LIN {X 0,Y 573.181,Z 132.082,A -85,B 0,C 180,E1 -2286.055,E2 -2286.055} C_VEL
LIN {X 0,Y 573.23,Z 132.081,A -85,B 0,C 180,E1 -2288.703,E2 -2288.703} C_VEL
LIN {X 0,Y 573.201,Z 132.082,A -85,B 0,C 180,E1 -2291.46,E2 -2291.46} C_VEL
LIN {X 0,Y 573.219,Z 132.079,A -85,B 0,C 180,E1 -2294.336,E2 -2294.336} C_VEL
LIN {X 0,Y 573.214,Z 132.079,A -85,B 0,C 180,E1 -2297.362,E2 -2297.362} C_VEL
LIN {X 0,Y 573.229,Z 132.08,A -85,B 0,C 180,E1 -2300.391,E2 -2300.391} C_VEL
LIN {X 0,Y 573.231,Z 132.078,A -85,B 0,C 180,E1 -2303.076,E2 -2303.076} C_VEL
LIN {X 0,Y 573.248,Z 132.074,A -85,B 0,C 180,E1 -2305.67,E2 -2305.67} C_VEL
LIN {X 0,Y 573.227,Z 132.081,A -85,B 0,C 180,E1 -2308.184,E2 -2308.184} C_VEL
LIN {X 0,Y 573.219,Z 132.083,A -85,B 0,C 180,E1 -2310.632,E2 -2310.632} C_VEL
LIN {X 0,Y 573.207,Z 132.079,A -85,B 0,C 180,E1 -2313.515,E2 -2313.515} C_VEL
LIN {X 0,Y 573.201,Z 132.087,A -85,B 0,C 180,E1 -2316.133,E2 -2316.133} C_VEL
LIN {X 0,Y 573.238,Z 132.076,A -85,B 0,C 180,E1 -2318.714,E2 -2318.714} C_VEL
LIN {X 0,Y 573.199,Z 132.08,A -85,B 0,C 180,E1 -2321.411,E2 -2321.411} C_VEL
LIN {X 0,Y 573.21,Z 132.084,A -85,B 0,C 180,E1 -2324.351,E2 -2324.351} C_VEL
LIN {X 0,Y 573.206,Z 132.081,A -85,B 0,C 180,E1 -2326.529,E2 -2326.529} C_VEL
LIN {X 0,Y 573.261,Z 132.075,A -85,B 0,C 180,E1 -2329.403,E2 -2329.403} C_VEL
LIN {X 0,Y 573.225,Z 132.081,A -85,B 0,C 180,E1 -2332.249,E2 -2332.249} C_VEL
LIN {X 0,Y 573.288,Z 132.07,A -85,B 0,C 180,E1 -2335.077,E2 -2335.077} C_VEL
LIN {X 0,Y 573.313,Z 132.072,A -85,B 0,C 180,E1 -2337.893,E2 -2337.893} C_VEL
LIN {X 0,Y 573.322,Z 132.07,A -85,B 0,C 180,E1 -2340,E2 -2340} C_VEL
LIN {X 0,Y 573.287,Z 132.071,A -85,B 0,C 180,E1 -2342.811,E2 -2342.811} C_VEL
LIN {X 0,Y 573.284,Z 132.078,A -85,B 0,C 180,E1 -2345.628,E2 -2345.628} C_VEL
LIN {X 0,Y 573.285,Z 132.18,A -85,B 0,C 180,E1 -2348.371,E2 -2348.371} C_VEL
LIN {X 0,Y 573.5,Z 140.017,A -85,B 0,C 180,E1 -2349.701,E2 -2349.701} C_VEL
LIN {X 0,Y 573.378,Z 155.55,A -85,B 0,C 180,E1 -2352.386,E2 -2352.386} C_VEL
LIN {X 0,Y 573.294,Z 166.446,A -85,B 0,C 180,E1 -2354.231,E2 -2354.231} C_VEL
LIN {X 0,Y 574.098,Z 171.713,A -85,B 0,C 180,E1 -2354.317,E2 -2354.317} C_VEL
LIN {X 0,Y 573.971,Z 236.172,A -85,B 0,C 180,E1 -2355.126,E2 -2355.126} C_VEL
LIN {X 0,Y 573.349,Z 242.014,A -85,B 0,C 180,E1 -2355.185,E2 -2355.185} C_VEL
LIN {X 0,Y 567.678,Z 260.997,A -85,B 0,C 180,E1 -2355.294,E2 -2355.294} C_VEL
LIN {X 0,Y 566.978,Z 266.837,A -85,B 0,C 180,E1 -2355.355,E2 -2355.355} C_VEL
LIN {X 0,Y 566.881,Z 279.861,A -85,B 0,C 180,E1 -2355.598,E2 -2355.598} C_VEL
LIN {X 0,Y 566.804,Z 291.142,A -85,B 0,C 180,E1 -2355.923,E2 -2355.923} C_VEL
LIN {X 0,Y 566.703,Z 302.843,A -85,B 0,C 180,E1 -2356.388,E2 -2356.388} C_VEL
LIN {X 0,Y 566.554,Z 313.939,A -85,B 0,C 180,E1 -2356.973,E2 -2356.973} C_VEL
LIN {X 0,Y 566.407,Z 324.984,A -85,B 0,C 180,E1 -2357.698,E2 -2357.698} C_VEL
LIN {X 0,Y 566.246,Z 335.181,A -85,B 0,C 180,E1 -2358.545,E2 -2358.545} C_VEL
LIN {X 0,Y 566.193,Z 343.437,A -85,B 0,C 180,E1 -2359.374,E2 -2359.374} C_VEL
LIN {X 0,Y 566.095,Z 351.459,A -85,B 0,C 180,E1 -2360.342,E2 -2360.342} C_VEL
LIN {X 0,Y 565.998,Z 358.286,A -85,B 0,C 180,E1 -2361.364,E2 -2361.364} C_VEL
LIN {X 0,Y 565.939,Z 363.21,A -85,B 0,C 180,E1 -2362.257,E2 -2362.257} C_VEL
LIN {X 0,Y 565.912,Z 368.377,A -85,B 0,C 180,E1 -2363.416,E2 -2363.416} C_VEL
LIN {X 0,Y 565.916,Z 372.21,A -85,B 0,C 180,E1 -2364.572,E2 -2364.572} C_VEL
LIN {X 0,Y 565.839,Z 374.92,A -85,B 0,C 180,E1 -2365.768,E2 -2365.768} C_VEL
LIN {X 0,Y 565.863,Z 376.12,A -85,B 0,C 180,E1 -2366.588,E2 -2366.588} C_VEL
LIN {X 0,Y 565.834,Z 376.788,A -85,B 0,C 180,E1 -2367.359,E2 -2367.359} C_VEL
LIN {X 0,Y 565.835,Z 376.98,A -85,B 0,C 180,E1 -2368.163,E2 -2368.163} C_VEL
LIN {X 0,Y 565.849,Z 376.658,A -85,B 0,C 180,E1 -2368.973,E2 -2368.973} C_VEL
LIN {X 0,Y 565.874,Z 375.805,A -85,B 0,C 180,E1 -2369.788,E2 -2369.788} C_VEL
LIN {X 0,Y 565.882,Z 373.468,A -85,B 0,C 180,E1 -2371.024,E2 -2371.024} C_VEL
LIN {X 0,Y 565.886,Z 369.468,A -85,B 0,C 180,E1 -2372.378,E2 -2372.378} C_VEL
LIN {X 0,Y 565.954,Z 363.904,A -85,B 0,C 180,E1 -2373.694,E2 -2373.694} C_VEL
LIN {X 0,Y 565.987,Z 357.645,A -85,B 0,C 180,E1 -2374.834,E2 -2374.834} C_VEL
LIN {X 0,Y 566.077,Z 349.885,A -85,B 0,C 180,E1 -2375.951,E2 -2375.951} C_VEL
LIN {X 0,Y 566.18,Z 341.688,A -85,B 0,C 180,E1 -2376.905,E2 -2376.905} C_VEL
LIN {X 0,Y 566.332,Z 332.526,A -85,B 0,C 180,E1 -2377.788,E2 -2377.788} C_VEL
LIN {X 0,Y 566.413,Z 322.247,A -85,B 0,C 180,E1 -2378.583,E2 -2378.583} C_VEL
LIN {X 0,Y 566.564,Z 311.758,A -85,B 0,C 180,E1 -2379.245,E2 -2379.245} C_VEL
LIN {X 0,Y 566.74,Z 300.242,A -85,B 0,C 180,E1 -2379.816,E2 -2379.816} C_VEL
LIN {X 0,Y 566.816,Z 288.611,A -85,B 0,C 180,E1 -2380.249,E2 -2380.249} C_VEL
LIN {X 0,Y 566.93,Z 275.731,A -85,B 0,C 180,E1 -2380.589,E2 -2380.589} C_VEL
LIN {X 0,Y 567.007,Z 254.604,A -85,B 0,C 180,E1 -2380.891,E2 -2380.891} C_VEL
LIN {X 0,Y 567.047,Z 170.943,A -85,B 0,C 180,E1 -2381.957,E2 -2381.957} C_VEL
LIN {X 0,Y 566.278,Z 166.148,A -85,B 0,C 180,E1 -2382.045,E2 -2382.045} C_VEL
LIN {X 0,Y 566.471,Z 147.947,A -85,B 0,C 180,E1 -2385.255,E2 -2385.255} C_VEL
LIN {X 0,Y 566.53,Z 135.587,A -85,B 0,C 180,E1 -2387.46,E2 -2387.46} C_VEL
LIN {X 0,Y 566.211,Z 132.957,A -85,B 0,C 180,E1 -2387.984,E2 -2387.984} C_VEL
LIN {X 0,Y 566.208,Z 132.959,A -85,B 0,C 180,E1 -2390.725,E2 -2390.725} C_VEL
LIN {X 0,Y 566.183,Z 132.954,A -85,B 0,C 180,E1 -2393.428,E2 -2393.428} C_VEL
LIN {X 0,Y 566.201,Z 132.957,A -85,B 0,C 180,E1 -2396.268,E2 -2396.268} C_VEL
LIN {X 0,Y 566.181,Z 132.956,A -85,B 0,C 180,E1 -2398.926,E2 -2398.926} C_VEL
LIN {X 0,Y 566.147,Z 132.96,A -85,B 0,C 180,E1 -2401.853,E2 -2401.853} C_VEL
LIN {X 0,Y 566.184,Z 132.961,A -85,B 0,C 180,E1 -2404.249,E2 -2404.249} C_VEL
LIN {X 0,Y 566.162,Z 132.959,A -85,B 0,C 180,E1 -2406.722,E2 -2406.722} C_VEL
LIN {X 0,Y 566.189,Z 132.954,A -85,B 0,C 180,E1 -2408.901,E2 -2408.901} C_VEL
LIN {X 0,Y 566.167,Z 132.955,A -85,B 0,C 180,E1 -2411.17,E2 -2411.17} C_VEL
LIN {X 0,Y 566.172,Z 132.965,A -85,B 0,C 180,E1 -2414.151,E2 -2414.151} C_VEL
LIN {X 0,Y 566.171,Z 132.96,A -85,B 0,C 180,E1 -2416.358,E2 -2416.358} C_VEL
LIN {X 0,Y 566.216,Z 132.95,A -85,B 0,C 180,E1 -2419.269,E2 -2419.269} C_VEL
LIN {X 0,Y 566.192,Z 132.959,A -85,B 0,C 180,E1 -2422.152,E2 -2422.152} C_VEL
LIN {X 0,Y 566.253,Z 132.944,A -85,B 0,C 180,E1 -2425.015,E2 -2425.015} C_VEL
LIN {X 0,Y 566.281,Z 132.951,A -85,B 0,C 180,E1 -2427.866,E2 -2427.866} C_VEL
LIN {X 0,Y 566.289,Z 132.947,A -85,B 0,C 180,E1 -2429.999,E2 -2429.999} C_VEL
LIN {X 0,Y 566.241,Z 132.946,A -85,B 0,C 180,E1 -2432.845,E2 -2432.845} C_VEL
LIN {X 0,Y 566.24,Z 132.956,A -85,B 0,C 180,E1 -2435.698,E2 -2435.698} C_VEL
LIN {X 0,Y 566.188,Z 132.953,A -85,B 0,C 180,E1 -2438.566,E2 -2438.566} C_VEL
LIN {X 0,Y 566.196,Z 132.96,A -85,B 0,C 180,E1 -2441.455,E2 -2441.455} C_VEL
LIN {X 0,Y 566.179,Z 132.954,A -85,B 0,C 180,E1 -2444.482,E2 -2444.482} C_VEL
LIN {X 0,Y 566.16,Z 132.964,A -85,B 0,C 180,E1 -2447.332,E2 -2447.332} C_VEL
LIN {X 0,Y 566.176,Z 132.961,A -85,B 0,C 180,E1 -2449.581,E2 -2449.581} C_VEL
LIN {X 0,Y 566.148,Z 132.96,A -85,B 0,C 180,E1 -2451.864,E2 -2451.864} C_VEL
LIN {X 0,Y 566.18,Z 132.959,A -85,B 0,C 180,E1 -2455.02,E2 -2455.02} C_VEL
LIN {X 0,Y 566.16,Z 132.964,A -85,B 0,C 180,E1 -2457.341,E2 -2457.341} C_VEL
LIN {X 0,Y 566.146,Z 132.96,A -85,B 0,C 180,E1 -2459.771,E2 -2459.771} C_VEL
LIN {X 0,Y 566.19,Z 132.953,A -85,B 0,C 180,E1 -2462.427,E2 -2462.427} C_VEL
LIN {X 0,Y 566.159,Z 132.965,A -85,B 0,C 180,E1 -2464.986,E2 -2464.986} C_VEL
LIN {X 0,Y 566.188,Z 132.956,A -85,B 0,C 180,E1 -2467.461,E2 -2467.461} C_VEL
LIN {X 0,Y 566.202,Z 132.951,A -85,B 0,C 180,E1 -2470.199,E2 -2470.199} C_VEL
LIN {X 0,Y 566.174,Z 132.962,A -85,B 0,C 180,E1 -2473.056,E2 -2473.056} C_VEL
LIN {X 0,Y 566.152,Z 132.957,A -85,B 0,C 180,E1 -2476.053,E2 -2476.053} C_VEL
LIN {X 0,Y 566.146,Z 132.967,A -85,B 0,C 180,E1 -2478.857,E2 -2478.857} C_VEL
LIN {X 0,Y 566.193,Z 132.953,A -85,B 0,C 180,E1 -2481.443,E2 -2481.443} C_VEL
LIN {X 0,Y 566.133,Z 132.963,A -85,B 0,C 180,E1 -2484.305,E2 -2484.305} C_VEL
LIN {X 0,Y 566.186,Z 132.958,A -85,B 0,C 180,E1 -2486.895,E2 -2486.895} C_VEL
LIN {X 0,Y 566.154,Z 132.957,A -85,B 0,C 180,E1 -2489.405,E2 -2489.405} C_VEL
LIN {X 0,Y 566.135,Z 132.96,A -85,B 0,C 180,E1 -2491.853,E2 -2491.853} C_VEL
LIN {X 0,Y 566.182,Z 132.959,A -85,B 0,C 180,E1 -2494.249,E2 -2494.249} C_VEL
LIN {X 0,Y 566.149,Z 132.962,A -85,B 0,C 180,E1 -2496.722,E2 -2496.722} C_VEL
LIN {X 0,Y 566.183,Z 132.956,A -85,B 0,C 180,E1 -2498.901,E2 -2498.901} C_VEL
LIN {X 0,Y 566.175,Z 132.954,A -85,B 0,C 180,E1 -2501.171,E2 -2501.171} C_VEL
LIN {X 0,Y 566.162,Z 132.964,A -85,B 0,C 180,E1 -2504.151,E2 -2504.151} C_VEL
LIN {X 0,Y 566.155,Z 132.964,A -85,B 0,C 180,E1 -2506.358,E2 -2506.358} C_VEL
LIN {X 0,Y 566.204,Z 132.951,A -85,B 0,C 180,E1 -2509.269,E2 -2509.269} C_VEL
LIN {X 0,Y 566.179,Z 132.963,A -85,B 0,C 180,E1 -2512.152,E2 -2512.152} C_VEL
LIN {X 0,Y 566.243,Z 132.946,A -85,B 0,C 180,E1 -2515.016,E2 -2515.016} C_VEL
LIN {X 0,Y 566.273,Z 132.95,A -85,B 0,C 180,E1 -2517.866,E2 -2517.866} C_VEL
LIN {X 0,Y 566.278,Z 132.95,A -85,B 0,C 180,E1 -2520,E2 -2520} C_VEL
LIN {X 0,Y 566.23,Z 132.947,A -85,B 0,C 180,E1 -2522.846,E2 -2522.846} C_VEL
LIN {X 0,Y 566.23,Z 132.955,A -85,B 0,C 180,E1 -2525.698,E2 -2525.698} C_VEL
LIN {X 0,Y 566.177,Z 132.954,A -85,B 0,C 180,E1 -2528.566,E2 -2528.566} C_VEL
LIN {X 0,Y 566.184,Z 132.959,A -85,B 0,C 180,E1 -2531.455,E2 -2531.455} C_VEL
LIN {X 0,Y 566.194,Z 132.952,A -85,B 0,C 180,E1 -2534.494,E2 -2534.494} C_VEL
LIN {X 0,Y 566.148,Z 132.963,A -85,B 0,C 180,E1 -2537.333,E2 -2537.333} C_VEL
LIN {X 0,Y 566.165,Z 132.965,A -85,B 0,C 180,E1 -2539.582,E2 -2539.582} C_VEL
LIN {X 0,Y 566.138,Z 132.963,A -85,B 0,C 180,E1 -2541.865,E2 -2541.865} C_VEL
LIN {X 0,Y 566.144,Z 132.959,A -85,B 0,C 180,E1 -2544.183,E2 -2544.183} C_VEL
LIN {X 0,Y 566.163,Z 132.956,A -85,B 0,C 180,E1 -2546.652,E2 -2546.652} C_VEL
LIN {X 0,Y 566.138,Z 132.962,A -85,B 0,C 180,E1 -2549.772,E2 -2549.772} C_VEL
LIN {X 0,Y 566.183,Z 132.953,A -85,B 0,C 180,E1 -2552.428,E2 -2552.428} C_VEL
LIN {X 0,Y 566.151,Z 132.963,A -85,B 0,C 180,E1 -2554.987,E2 -2554.987} C_VEL
LIN {X 0,Y 566.181,Z 132.958,A -85,B 0,C 180,E1 -2557.462,E2 -2557.462} C_VEL
LIN {X 0,Y 566.159,Z 132.956,A -85,B 0,C 180,E1 -2560.203,E2 -2560.203} C_VEL
LIN {X 0,Y 566.141,Z 132.968,A -85,B 0,C 180,E1 -2563.06,E2 -2563.06} C_VEL
LIN {X 0,Y 566.148,Z 132.957,A -85,B 0,C 180,E1 -2566.054,E2 -2566.054} C_VEL
LIN {X 0,Y 566.136,Z 132.968,A -85,B 0,C 180,E1 -2568.858,E2 -2568.858} C_VEL
LIN {X 0,Y 566.165,Z 132.956,A -85,B 0,C 180,E1 -2571.636,E2 -2571.636} C_VEL
LIN {X 0,Y 566.126,Z 132.963,A -85,B 0,C 180,E1 -2574.306,E2 -2574.306} C_VEL
LIN {X 0,Y 566.158,Z 132.964,A -85,B 0,C 180,E1 -2576.895,E2 -2576.895} C_VEL
LIN {X 0,Y 566.145,Z 132.959,A -85,B 0,C 180,E1 -2579.406,E2 -2579.406} C_VEL
LIN {X 0,Y 566.137,Z 132.96,A -85,B 0,C 180,E1 -2581.854,E2 -2581.854} C_VEL
LIN {X 0,Y 566.172,Z 132.96,A -85,B 0,C 180,E1 -2584.25,E2 -2584.25} C_VEL
LIN {X 0,Y 566.157,Z 133.092,A -85,B 0,C 180,E1 -2586.833,E2 -2586.833} C_VEL
LIN {X 0,Y 566.94,Z 137.904,A -85,B 0,C 180,E1 -2587.593,E2 -2587.593} C_VEL
LIN {X 0,Y 566.776,Z 155.695,A -85,B 0,C 180,E1 -2590.252,E2 -2590.252} C_VEL
LIN {X 0,Y 566.546,Z 172.893,A -85,B 0,C 180,E1 -2592.782,E2 -2592.782} C_VEL
LIN {X 0,Y 566.404,Z 192.436,A -85,B 0,C 180,E1 -2595.632,E2 -2595.632} C_VEL
LIN {X 0,Y 566.421,Z 195.196,A -85,B 0,C 180,E1 -2595.999,E2 -2595.999} C_VEL
LIN {X 0,Y 567.174,Z 201.344,A -85,B 0,C 180,E1 -2596.097,E2 -2596.097} C_VEL
LIN {X 0,Y 566.965,Z 302.98,A -85,B 0,C 180,E1 -2597.404,E2 -2597.404} C_VEL
LIN {X 0,Y 566.839,Z 316.24,A -85,B 0,C 180,E1 -2597.719,E2 -2597.719} C_VEL
LIN {X 0,Y 566.741,Z 328.394,A -85,B 0,C 180,E1 -2598.149,E2 -2598.149} C_VEL
LIN {X 0,Y 566.602,Z 340.372,A -85,B 0,C 180,E1 -2598.72,E2 -2598.72} C_VEL
LIN {X 0,Y 566.439,Z 352.205,A -85,B 0,C 180,E1 -2599.456,E2 -2599.456} C_VEL
LIN {X 0,Y 566.325,Z 362.612,A -85,B 0,C 180,E1 -2600.266,E2 -2600.266} C_VEL
LIN {X 0,Y 566.207,Z 371.119,A -85,B 0,C 180,E1 -2601.075,E2 -2601.075} C_VEL
LIN {X 0,Y 566.112,Z 378.966,A -85,B 0,C 180,E1 -2601.972,E2 -2601.972} C_VEL
LIN {X 0,Y 566.003,Z 386.627,A -85,B 0,C 180,E1 -2603.047,E2 -2603.047} C_VEL
LIN {X 0,Y 566.004,Z 393.683,A -85,B 0,C 180,E1 -2604.3,E2 -2604.3} C_VEL
LIN {X 0,Y 565.933,Z 398.375,A -85,B 0,C 180,E1 -2605.371,E2 -2605.371} C_VEL
LIN {X 0,Y 565.927,Z 401.96,A -85,B 0,C 180,E1 -2606.441,E2 -2606.441} C_VEL
LIN {X 0,Y 565.877,Z 403.809,A -85,B 0,C 180,E1 -2607.153,E2 -2607.153} C_VEL
LIN {X 0,Y 565.846,Z 406.185,A -85,B 0,C 180,E1 -2608.577,E2 -2608.577} C_VEL
LIN {X 0,Y 565.839,Z 407,A -85,B 0,C 180,E1 -2610.001,E2 -2610.001} C_VEL
LIN {X 0,Y 565.846,Z 406.184,A -85,B 0,C 180,E1 -2611.424,E2 -2611.424} C_VEL
LIN {X 0,Y 565.878,Z 403.809,A -85,B 0,C 180,E1 -2612.848,E2 -2612.848} C_VEL
LIN {X 0,Y 565.926,Z 400.894,A -85,B 0,C 180,E1 -2613.917,E2 -2613.917} C_VEL
LIN {X 0,Y 565.878,Z 396.946,A -85,B 0,C 180,E1 -2614.988,E2 -2614.988} C_VEL
LIN {X 0,Y 566.002,Z 391.864,A -85,B 0,C 180,E1 -2616.059,E2 -2616.059} C_VEL
LIN {X 0,Y 566.041,Z 385.463,A -85,B 0,C 180,E1 -2617.133,E2 -2617.133} C_VEL
LIN {X 0,Y 566.134,Z 377.473,A -85,B 0,C 180,E1 -2618.208,E2 -2618.208} C_VEL
LIN {X 0,Y 566.229,Z 369.328,A -85,B 0,C 180,E1 -2619.106,E2 -2619.106} C_VEL
LIN {X 0,Y 566.348,Z 359.392,A -85,B 0,C 180,E1 -2620.005,E2 -2620.005} C_VEL
LIN {X 0,Y 566.536,Z 348.282,A -85,B 0,C 180,E1 -2620.808,E2 -2620.808} C_VEL
LIN {X 0,Y 566.614,Z 337.161,A -85,B 0,C 180,E1 -2621.447,E2 -2621.447} C_VEL
LIN {X 0,Y 566.746,Z 324.964,A -85,B 0,C 180,E1 -2621.989,E2 -2621.989} C_VEL
LIN {X 0,Y 566.918,Z 312.151,A -85,B 0,C 180,E1 -2622.394,E2 -2622.394} C_VEL
LIN {X 0,Y 566.994,Z 300.066,A -85,B 0,C 180,E1 -2622.642,E2 -2622.642} C_VEL
LIN {X 0,Y 567.043,Z 199.346,A -85,B 0,C 180,E1 -2623.932,E2 -2623.932} C_VEL
LIN {X 0,Y 566.385,Z 194.788,A -85,B 0,C 180,E1 -2624.026,E2 -2624.026} C_VEL
LIN {X 0,Y 566.532,Z 175.015,A -85,B 0,C 180,E1 -2626.896,E2 -2626.896} C_VEL
LIN {X 0,Y 566.723,Z 157.67,A -85,B 0,C 180,E1 -2629.424,E2 -2629.424} C_VEL
LIN {X 0,Y 566.911,Z 139.991,A -85,B 0,C 180,E1 -2632.025,E2 -2632.025} C_VEL
LIN {X 0,Y 566.504,Z 134.839,A -85,B 0,C 180,E1 -2632.799,E2 -2632.799} C_VEL
LIN {X 0,Y 566.155,Z 132.966,A -85,B 0,C 180,E1 -2633.093,E2 -2633.093} C_VEL
LIN {X 0,Y 566.173,Z 132.961,A -85,B 0,C 180,E1 -2635.752,E2 -2635.752} C_VEL
LIN {X 0,Y 566.14,Z 132.96,A -85,B 0,C 180,E1 -2638.19,E2 -2638.19} C_VEL
LIN {X 0,Y 566.172,Z 132.963,A -85,B 0,C 180,E1 -2641.073,E2 -2641.073} C_VEL
LIN {X 0,Y 566.198,Z 132.954,A -85,B 0,C 180,E1 -2643.732,E2 -2643.732} C_VEL
LIN {X 0,Y 566.148,Z 132.961,A -85,B 0,C 180,E1 -2646.574,E2 -2646.574} C_VEL
LIN {X 0,Y 566.205,Z 132.956,A -85,B 0,C 180,E1 -2649.275,E2 -2649.275} C_VEL
LIN {X 0,Y 566.146,Z 132.958,A -85,B 0,C 180,E1 -2652.094,E2 -2652.094} C_VEL
LIN {X 0,Y 566.167,Z 132.961,A -85,B 0,C 180,E1 -2655.037,E2 -2655.037} C_VEL
LIN {X 0,Y 566.146,Z 132.958,A -85,B 0,C 180,E1 -2657.906,E2 -2657.906} C_VEL
LIN {X 0,Y 566.205,Z 132.959,A -85,B 0,C 180,E1 -2660.726,E2 -2660.726} C_VEL
LIN {X 0,Y 566.181,Z 132.954,A -85,B 0,C 180,E1 -2663.429,E2 -2663.429} C_VEL
LIN {X 0,Y 566.198,Z 132.957,A -85,B 0,C 180,E1 -2666.269,E2 -2666.269} C_VEL
LIN {X 0,Y 566.183,Z 132.956,A -85,B 0,C 180,E1 -2668.926,E2 -2668.926} C_VEL
LIN {X 0,Y 566.145,Z 132.96,A -85,B 0,C 180,E1 -2671.854,E2 -2671.854} C_VEL
LIN {X 0,Y 566.193,Z 132.961,A -85,B 0,C 180,E1 -2674.25,E2 -2674.25} C_VEL
LIN {X 0,Y 566.163,Z 132.956,A -85,B 0,C 180,E1 -2677.368,E2 -2677.368} C_VEL
LIN {X 0,Y 566.173,Z 132.956,A -85,B 0,C 180,E1 -2679.661,E2 -2679.661} C_VEL
LIN {X 0,Y 566.169,Z 132.962,A -85,B 0,C 180,E1 -2681.921,E2 -2681.921} C_VEL
LIN {X 0,Y 566.187,Z 132.954,A -85,B 0,C 180,E1 -2684.89,E2 -2684.89} C_VEL
LIN {X 0,Y 566.184,Z 132.961,A -85,B 0,C 180,E1 -2687.818,E2 -2687.818} C_VEL
LIN {X 0,Y 566.17,Z 132.965,A -85,B 0,C 180,E1 -2689.992,E2 -2689.992} C_VEL
LIN {X 0,Y 566.194,Z 132.958,A -85,B 0,C 180,E1 -2692.152,E2 -2692.152} C_VEL
LIN {X 0,Y 566.263,Z 132.945,A -85,B 0,C 180,E1 -2695.016,E2 -2695.016} C_VEL
LIN {X 0,Y 566.283,Z 132.949,A -85,B 0,C 180,E1 -2697.866,E2 -2697.866} C_VEL
LIN {X 0,Y 566.291,Z 132.946,A -85,B 0,C 180,E1 -2700,E2 -2700} C_VEL
LIN {X 0,Y 566.256,Z 132.947,A -85,B 0,C 180,E1 -2702.846,E2 -2702.846} C_VEL
LIN {X 0,Y 566.252,Z 132.953,A -85,B 0,C 180,E1 -2705.699,E2 -2705.699} C_VEL
LIN {X 0,Y 566.265,Z 133.144,A -85,B 0,C 180,E1 -2708.341,E2 -2708.341} C_VEL
LIN {X 0,Y 566.445,Z 141.838,A -85,B 0,C 180,E1 -2709.823,E2 -2709.823} C_VEL
LIN {X 0,Y 566.37,Z 158.639,A -85,B 0,C 180,E1 -2712.724,E2 -2712.724} C_VEL
LIN {X 0,Y 566.241,Z 166.201,A -85,B 0,C 180,E1 -2714.052,E2 -2714.052} C_VEL
LIN {X 0,Y 567.214,Z 173.101,A -85,B 0,C 180,E1 -2714.165,E2 -2714.165} C_VEL
LIN {X 0,Y 566.978,Z 266.837,A -85,B 0,C 180,E1 -2715.355,E2 -2715.355} C_VEL
LIN {X 0,Y 566.292,Z 270.755,A -85,B 0,C 180,E1 -2715.396,E2 -2715.396} C_VEL
LIN {X 0,Y 563.478,Z 276.89,A -85,B 0,C 180,E1 -2715.444,E2 -2715.444} C_VEL
LIN {X 0,Y 560.627,Z 282.948,A -85,B 0,C 180,E1 -2715.528,E2 -2715.528} C_VEL
LIN {X 0,Y 559.881,Z 286.741,A -85,B 0,C 180,E1 -2715.627,E2 -2715.627} C_VEL
LIN {X 0,Y 559.804,Z 297.991,A -85,B 0,C 180,E1 -2716.034,E2 -2716.034} C_VEL
LIN {X 0,Y 559.64,Z 309.982,A -85,B 0,C 180,E1 -2716.601,E2 -2716.601} C_VEL
LIN {X 0,Y 559.437,Z 321.167,A -85,B 0,C 180,E1 -2717.299,E2 -2717.299} C_VEL
LIN {X 0,Y 559.33,Z 330.659,A -85,B 0,C 180,E1 -2718.024,E2 -2718.024} C_VEL
LIN {X 0,Y 559.18,Z 339.934,A -85,B 0,C 180,E1 -2718.883,E2 -2718.883} C_VEL
LIN {X 0,Y 559.056,Z 348.31,A -85,B 0,C 180,E1 -2719.842,E2 -2719.842} C_VEL
LIN {X 0,Y 558.969,Z 355.321,A -85,B 0,C 180,E1 -2720.805,E2 -2720.805} C_VEL
LIN {X 0,Y 558.891,Z 361.221,A -85,B 0,C 180,E1 -2721.787,E2 -2721.787} C_VEL
LIN {X 0,Y 558.821,Z 366.699,A -85,B 0,C 180,E1 -2722.947,E2 -2722.947} C_VEL
LIN {X 0,Y 558.808,Z 371.006,A -85,B 0,C 180,E1 -2724.126,E2 -2724.126} C_VEL
LIN {X 0,Y 558.763,Z 374.146,A -85,B 0,C 180,E1 -2725.319,E2 -2725.319} C_VEL
LIN {X 0,Y 558.743,Z 375.579,A -85,B 0,C 180,E1 -2726.119,E2 -2726.119} C_VEL
LIN {X 0,Y 558.751,Z 376.492,A -85,B 0,C 180,E1 -2726.924,E2 -2726.924} C_VEL
LIN {X 0,Y 558.751,Z 376.936,A -85,B 0,C 180,E1 -2728.301,E2 -2728.301} C_VEL
LIN {X 0,Y 558.774,Z 375.825,A -85,B 0,C 180,E1 -2729.79,E2 -2729.79} C_VEL
LIN {X 0,Y 558.821,Z 373.069,A -85,B 0,C 180,E1 -2731.217,E2 -2731.217} C_VEL
LIN {X 0,Y 558.819,Z 370.128,A -85,B 0,C 180,E1 -2732.231,E2 -2732.231} C_VEL
LIN {X 0,Y 558.845,Z 366.608,A -85,B 0,C 180,E1 -2733.165,E2 -2733.165} C_VEL
LIN {X 0,Y 558.882,Z 360.306,A -85,B 0,C 180,E1 -2734.464,E2 -2734.464} C_VEL
LIN {X 0,Y 558.969,Z 353.456,A -85,B 0,C 180,E1 -2735.557,E2 -2735.557} C_VEL
LIN {X 0,Y 559.103,Z 345.975,A -85,B 0,C 180,E1 -2736.541,E2 -2736.541} C_VEL
LIN {X 0,Y 559.234,Z 336.904,A -85,B 0,C 180,E1 -2737.502,E2 -2737.502} C_VEL
LIN {X 0,Y 559.318,Z 328.628,A -85,B 0,C 180,E1 -2738.232,E2 -2738.232} C_VEL
LIN {X 0,Y 559.466,Z 317.774,A -85,B 0,C 180,E1 -2739.026,E2 -2739.026} C_VEL
LIN {X 0,Y 559.635,Z 306.79,A -85,B 0,C 180,E1 -2739.652,E2 -2739.652} C_VEL
LIN {X 0,Y 559.827,Z 296.713,A -85,B 0,C 180,E1 -2740.109,E2 -2740.109} C_VEL
LIN {X 0,Y 559.946,Z 283.908,A -85,B 0,C 180,E1 -2740.548,E2 -2740.548} C_VEL
LIN {X 0,Y 560.037,Z 271.434,A -85,B 0,C 180,E1 -2740.819,E2 -2740.819} C_VEL
LIN {X 0,Y 560.26,Z 172.217,A -85,B 0,C 180,E1 -2742.114,E2 -2742.114} C_VEL
LIN {X 0,Y 559.258,Z 166.242,A -85,B 0,C 180,E1 -2742.227,E2 -2742.227} C_VEL
LIN {X 0,Y 559.49,Z 147.656,A -85,B 0,C 180,E1 -2745.545,E2 -2745.545} C_VEL
LIN {X 0,Y 559.486,Z 136.152,A -85,B 0,C 180,E1 -2747.62,E2 -2747.62} C_VEL
LIN {X 0,Y 559.17,Z 133.835,A -85,B 0,C 180,E1 -2748.08,E2 -2748.08} C_VEL
LIN {X 0,Y 559.172,Z 133.829,A -85,B 0,C 180,E1 -2751.193,E2 -2751.193} C_VEL
LIN {X 0,Y 559.121,Z 133.834,A -85,B 0,C 180,E1 -2753.787,E2 -2753.787} C_VEL
LIN {X 0,Y 559.15,Z 133.838,A -85,B 0,C 180,E1 -2756.424,E2 -2756.424} C_VEL
LIN {X 0,Y 559.146,Z 133.832,A -85,B 0,C 180,E1 -2758.98,E2 -2758.98} C_VEL
LIN {X 0,Y 559.109,Z 133.835,A -85,B 0,C 180,E1 -2761.631,E2 -2761.631} C_VEL
LIN {X 0,Y 559.153,Z 133.832,A -85,B 0,C 180,E1 -2763.901,E2 -2763.901} C_VEL
LIN {X 0,Y 559.101,Z 133.836,A -85,B 0,C 180,E1 -2767.065,E2 -2767.065} C_VEL
LIN {X 0,Y 559.117,Z 133.834,A -85,B 0,C 180,E1 -2769.392,E2 -2769.392} C_VEL
LIN {X 0,Y 559.109,Z 133.837,A -85,B 0,C 180,E1 -2771.684,E2 -2771.684} C_VEL
LIN {X 0,Y 559.132,Z 133.833,A -85,B 0,C 180,E1 -2774.694,E2 -2774.694} C_VEL
LIN {X 0,Y 559.146,Z 133.833,A -85,B 0,C 180,E1 -2777.662,E2 -2777.662} C_VEL
LIN {X 0,Y 559.122,Z 133.84,A -85,B 0,C 180,E1 -2779.864,E2 -2779.864} C_VEL
LIN {X 0,Y 559.154,Z 133.829,A -85,B 0,C 180,E1 -2782.779,E2 -2782.779} C_VEL
LIN {X 0,Y 559.23,Z 133.819,A -85,B 0,C 180,E1 -2784.953,E2 -2784.953} C_VEL
LIN {X 0,Y 559.252,Z 133.826,A -85,B 0,C 180,E1 -2787.839,E2 -2787.839} C_VEL
LIN {X 0,Y 559.258,Z 133.823,A -85,B 0,C 180,E1 -2789.999,E2 -2789.999} C_VEL
LIN {X 0,Y 559.21,Z 133.822,A -85,B 0,C 180,E1 -2792.881,E2 -2792.881} C_VEL
LIN {X 0,Y 559.208,Z 133.831,A -85,B 0,C 180,E1 -2795.77,E2 -2795.77} C_VEL
LIN {X 0,Y 559.154,Z 133.829,A -85,B 0,C 180,E1 -2798.674,E2 -2798.674} C_VEL
LIN {X 0,Y 559.157,Z 133.838,A -85,B 0,C 180,E1 -2801.601,E2 -2801.601} C_VEL
LIN {X 0,Y 559.156,Z 133.829,A -85,B 0,C 180,E1 -2804.575,E2 -2804.575} C_VEL
LIN {X 0,Y 559.115,Z 133.842,A -85,B 0,C 180,E1 -2807.558,E2 -2807.558} C_VEL
LIN {X 0,Y 559.139,Z 133.834,A -85,B 0,C 180,E1 -2809.838,E2 -2809.838} C_VEL
LIN {X 0,Y 559.103,Z 133.835,A -85,B 0,C 180,E1 -2812.154,E2 -2812.154} C_VEL
LIN {X 0,Y 559.139,Z 133.839,A -85,B 0,C 180,E1 -2815.177,E2 -2815.177} C_VEL
LIN {X 0,Y 559.101,Z 133.838,A -85,B 0,C 180,E1 -2817.716,E2 -2817.716} C_VEL
LIN {X 0,Y 559.092,Z 133.836,A -85,B 0,C 180,E1 -2820.186,E2 -2820.186} C_VEL
LIN {X 0,Y 559.146,Z 133.833,A -85,B 0,C 180,E1 -2822.715,E2 -2822.715} C_VEL
LIN {X 0,Y 559.111,Z 133.84,A -85,B 0,C 180,E1 -2825.324,E2 -2825.324} C_VEL
LIN {X 0,Y 559.123,Z 133.833,A -85,B 0,C 180,E1 -2828.017,E2 -2828.017} C_VEL
LIN {X 0,Y 559.123,Z 133.84,A -85,B 0,C 180,E1 -2830.814,E2 -2830.814} C_VEL
LIN {X 0,Y 559.103,Z 133.835,A -85,B 0,C 180,E1 -2833.737,E2 -2833.737} C_VEL
LIN {X 0,Y 559.103,Z 133.837,A -85,B 0,C 180,E1 -2836.262,E2 -2836.262} C_VEL
LIN {X 0,Y 559.11,Z 133.838,A -85,B 0,C 180,E1 -2839.183,E2 -2839.183} C_VEL
LIN {X 0,Y 559.162,Z 133.831,A -85,B 0,C 180,E1 -2841.192,E2 -2841.192} C_VEL
LIN {X 0,Y 559.111,Z 133.834,A -85,B 0,C 180,E1 -2843.787,E2 -2843.787} C_VEL
LIN {X 0,Y 559.138,Z 133.837,A -85,B 0,C 180,E1 -2846.423,E2 -2846.423} C_VEL
LIN {X 0,Y 559.139,Z 133.834,A -85,B 0,C 180,E1 -2848.979,E2 -2848.979} C_VEL
LIN {X 0,Y 559.097,Z 133.836,A -85,B 0,C 180,E1 -2851.631,E2 -2851.631} C_VEL
LIN {X 0,Y 559.147,Z 133.831,A -85,B 0,C 180,E1 -2853.901,E2 -2853.901} C_VEL
LIN {X 0,Y 559.098,Z 133.843,A -85,B 0,C 180,E1 -2856.58,E2 -2856.58} C_VEL
LIN {X 0,Y 559.14,Z 133.83,A -85,B 0,C 180,E1 -2859.394,E2 -2859.394} C_VEL
LIN {X 0,Y 559.106,Z 133.836,A -85,B 0,C 180,E1 -2861.684,E2 -2861.684} C_VEL
LIN {X 0,Y 559.12,Z 133.836,A -85,B 0,C 180,E1 -2864.694,E2 -2864.694} C_VEL
LIN {X 0,Y 559.138,Z 133.833,A -85,B 0,C 180,E1 -2867.662,E2 -2867.662} C_VEL
LIN {X 0,Y 559.113,Z 133.839,A -85,B 0,C 180,E1 -2869.864,E2 -2869.864} C_VEL
LIN {X 0,Y 559.14,Z 133.831,A -85,B 0,C 180,E1 -2872.779,E2 -2872.779} C_VEL
LIN {X 0,Y 559.22,Z 133.821,A -85,B 0,C 180,E1 -2874.953,E2 -2874.953} C_VEL
LIN {X 0,Y 559.243,Z 133.825,A -85,B 0,C 180,E1 -2877.839,E2 -2877.839} C_VEL
LIN {X 0,Y 559.246,Z 133.826,A -85,B 0,C 180,E1 -2880,E2 -2880} C_VEL
LIN {X 0,Y 559.198,Z 133.823,A -85,B 0,C 180,E1 -2882.881,E2 -2882.881} C_VEL
LIN {X 0,Y 559.199,Z 133.832,A -85,B 0,C 180,E1 -2885.77,E2 -2885.77} C_VEL
LIN {X 0,Y 559.142,Z 133.83,A -85,B 0,C 180,E1 -2888.675,E2 -2888.675} C_VEL
LIN {X 0,Y 559.146,Z 133.838,A -85,B 0,C 180,E1 -2891.602,E2 -2891.602} C_VEL
LIN {X 0,Y 559.144,Z 133.83,A -85,B 0,C 180,E1 -2894.576,E2 -2894.576} C_VEL
LIN {X 0,Y 559.103,Z 133.845,A -85,B 0,C 180,E1 -2897.559,E2 -2897.559} C_VEL
LIN {X 0,Y 559.128,Z 133.837,A -85,B 0,C 180,E1 -2899.839,E2 -2899.839} C_VEL
LIN {X 0,Y 559.093,Z 133.837,A -85,B 0,C 180,E1 -2902.155,E2 -2902.155} C_VEL
LIN {X 0,Y 559.13,Z 133.838,A -85,B 0,C 180,E1 -2905.178,E2 -2905.178} C_VEL
LIN {X 0,Y 559.092,Z 133.841,A -85,B 0,C 180,E1 -2907.717,E2 -2907.717} C_VEL
LIN {X 0,Y 559.084,Z 133.838,A -85,B 0,C 180,E1 -2910.187,E2 -2910.187} C_VEL
LIN {X 0,Y 559.138,Z 133.833,A -85,B 0,C 180,E1 -2912.716,E2 -2912.716} C_VEL
LIN {X 0,Y 559.104,Z 133.843,A -85,B 0,C 180,E1 -2915.326,E2 -2915.326} C_VEL
LIN {X 0,Y 559.115,Z 133.834,A -85,B 0,C 180,E1 -2918.019,E2 -2918.019} C_VEL
LIN {X 0,Y 559.095,Z 133.841,A -85,B 0,C 180,E1 -2920.818,E2 -2920.818} C_VEL
LIN {X 0,Y 559.094,Z 133.837,A -85,B 0,C 180,E1 -2923.739,E2 -2923.739} C_VEL
LIN {X 0,Y 559.094,Z 133.837,A -85,B 0,C 180,E1 -2926.263,E2 -2926.263} C_VEL
LIN {X 0,Y 559.095,Z 133.842,A -85,B 0,C 180,E1 -2929.183,E2 -2929.183} C_VEL
LIN {X 0,Y 559.116,Z 133.834,A -85,B 0,C 180,E1 -2931.982,E2 -2931.982} C_VEL
LIN {X 0,Y 559.111,Z 133.844,A -85,B 0,C 180,E1 -2934.79,E2 -2934.79} C_VEL
LIN {X 0,Y 559.134,Z 133.833,A -85,B 0,C 180,E1 -2937.368,E2 -2937.368} C_VEL
LIN {X 0,Y 559.092,Z 133.839,A -85,B 0,C 180,E1 -2940.153,E2 -2940.153} C_VEL
LIN {X 0,Y 559.108,Z 133.838,A -85,B 0,C 180,E1 -2943.186,E2 -2943.186} C_VEL
LIN {X 0,Y 559.092,Z 133.84,A -85,B 0,C 180,E1 -2945.493,E2 -2945.493} C_VEL
LIN {X 0,Y 559.135,Z 134.04,A -85,B 0,C 180,E1 -2946.695,E2 -2946.695} C_VEL
LIN {X 0,Y 560.004,Z 140.304,A -85,B 0,C 180,E1 -2947.69,E2 -2947.69} C_VEL
LIN {X 0,Y 559.812,Z 158.472,A -85,B 0,C 180,E1 -2950.433,E2 -2950.433} C_VEL
LIN {X 0,Y 559.536,Z 177.141,A -85,B 0,C 180,E1 -2953.209,E2 -2953.209} C_VEL
LIN {X 0,Y 559.367,Z 194.91,A -85,B 0,C 180,E1 -2955.819,E2 -2955.819} C_VEL
LIN {X 0,Y 560.27,Z 202.149,A -85,B 0,C 180,E1 -2955.935,E2 -2955.935} C_VEL
LIN {X 0,Y 560.038,Z 302.979,A -85,B 0,C 180,E1 -2957.245,E2 -2957.245} C_VEL
LIN {X 0,Y 559.913,Z 316.239,A -85,B 0,C 180,E1 -2957.565,E2 -2957.565} C_VEL
LIN {X 0,Y 559.79,Z 328.393,A -85,B 0,C 180,E1 -2958,E2 -2958} C_VEL
LIN {X 0,Y 559.627,Z 340.204,A -85,B 0,C 180,E1 -2958.568,E2 -2958.568} C_VEL
LIN {X 0,Y 559.458,Z 352.202,A -85,B 0,C 180,E1 -2959.323,E2 -2959.323} C_VEL
LIN {X 0,Y 559.305,Z 362.613,A -85,B 0,C 180,E1 -2960.143,E2 -2960.143} C_VEL
LIN {X 0,Y 559.161,Z 371.12,A -85,B 0,C 180,E1 -2960.961,E2 -2960.961} C_VEL
LIN {X 0,Y 559.049,Z 378.966,A -85,B 0,C 180,E1 -2961.87,E2 -2961.87} C_VEL
LIN {X 0,Y 558.943,Z 386.627,A -85,B 0,C 180,E1 -2962.959,E2 -2962.959} C_VEL
LIN {X 0,Y 558.935,Z 393.683,A -85,B 0,C 180,E1 -2964.227,E2 -2964.227} C_VEL
LIN {X 0,Y 558.826,Z 398.375,A -85,B 0,C 180,E1 -2965.312,E2 -2965.312} C_VEL
LIN {X 0,Y 558.836,Z 401.96,A -85,B 0,C 180,E1 -2966.395,E2 -2966.395} C_VEL
LIN {X 0,Y 558.799,Z 403.808,A -85,B 0,C 180,E1 -2967.117,E2 -2967.117} C_VEL
LIN {X 0,Y 558.745,Z 406.184,A -85,B 0,C 180,E1 -2968.559,E2 -2968.559} C_VEL
LIN {X 0,Y 558.74,Z 407,A -85,B 0,C 180,E1 -2970.001,E2 -2970.001} C_VEL
LIN {X 0,Y 558.745,Z 406.183,A -85,B 0,C 180,E1 -2971.442,E2 -2971.442} C_VEL
LIN {X 0,Y 558.799,Z 403.809,A -85,B 0,C 180,E1 -2972.884,E2 -2972.884} C_VEL
LIN {X 0,Y 558.844,Z 400.893,A -85,B 0,C 180,E1 -2973.967,E2 -2973.967} C_VEL
LIN {X 0,Y 558.798,Z 396.946,A -85,B 0,C 180,E1 -2975.051,E2 -2975.051} C_VEL
LIN {X 0,Y 558.922,Z 391.864,A -85,B 0,C 180,E1 -2976.136,E2 -2976.136} C_VEL
LIN {X 0,Y 558.978,Z 385.463,A -85,B 0,C 180,E1 -2977.223,E2 -2977.223} C_VEL
LIN {X 0,Y 559.099,Z 377.472,A -85,B 0,C 180,E1 -2978.312,E2 -2978.312} C_VEL
LIN {X 0,Y 559.195,Z 369.327,A -85,B 0,C 180,E1 -2979.222,E2 -2979.222} C_VEL
LIN {X 0,Y 559.358,Z 359.39,A -85,B 0,C 180,E1 -2980.132,E2 -2980.132} C_VEL
LIN {X 0,Y 559.556,Z 348.387,A -85,B 0,C 180,E1 -2980.937,E2 -2980.937} C_VEL
LIN {X 0,Y 559.672,Z 336.445,A -85,B 0,C 180,E1 -2981.628,E2 -2981.628} C_VEL
LIN {X 0,Y 559.823,Z 324.961,A -85,B 0,C 180,E1 -2982.139,E2 -2982.139} C_VEL
LIN {X 0,Y 559.982,Z 312.149,A -85,B 0,C 180,E1 -2982.55,E2 -2982.55} C_VEL
LIN {X 0,Y 560.089,Z 298.555,A -85,B 0,C 180,E1 -2982.824,E2 -2982.824} C_VEL
LIN {X 0,Y 560.086,Z 199.699,A -85,B 0,C 180,E1 -2984.1,E2 -2984.1} C_VEL
LIN {X 0,Y 559.36,Z 194.81,A -85,B 0,C 180,E1 -2984.183,E2 -2984.183} C_VEL
LIN {X 0,Y 559.524,Z 175.089,A -85,B 0,C 180,E1 -2987.063,E2 -2987.063} C_VEL
LIN {X 0,Y 559.766,Z 157.426,A -85,B 0,C 180,E1 -2989.67,E2 -2989.67} C_VEL
LIN {X 0,Y 559.942,Z 139.643,A -85,B 0,C 180,E1 -2992.314,E2 -2992.314} C_VEL
LIN {X 0,Y 559.111,Z 133.844,A -85,B 0,C 180,E1 -2993.218,E2 -2993.218} C_VEL
LIN {X 0,Y 559.143,Z 133.834,A -85,B 0,C 180,E1 -2996.1,E2 -2996.1} C_VEL
LIN {X 0,Y 559.1,Z 133.838,A -85,B 0,C 180,E1 -2998.534,E2 -2998.534} C_VEL
LIN {X 0,Y 559.12,Z 133.843,A -85,B 0,C 180,E1 -3001.268,E2 -3001.268} C_VEL
LIN {X 0,Y 559.153,Z 133.83,A -85,B 0,C 180,E1 -3003.947,E2 -3003.947} C_VEL
LIN {X 0,Y 559.119,Z 133.842,A -85,B 0,C 180,E1 -3007.111,E2 -3007.111} C_VEL
LIN {X 0,Y 559.157,Z 133.829,A -85,B 0,C 180,E1 -3009.941,E2 -3009.941} C_VEL
LIN {X 0,Y 559.125,Z 133.837,A -85,B 0,C 180,E1 -3013.194,E2 -3013.194} C_VEL
LIN {X 0,Y 559.126,Z 133.832,A -85,B 0,C 180,E1 -3015.764,E2 -3015.764} C_VEL
LIN {X 0,Y 559.102,Z 133.837,A -85,B 0,C 180,E1 -3018.224,E2 -3018.224} C_VEL
LIN {X 0,Y 559.169,Z 133.829,A -85,B 0,C 180,E1 -3021.193,E2 -3021.193} C_VEL
LIN {X 0,Y 559.118,Z 133.833,A -85,B 0,C 180,E1 -3023.788,E2 -3023.788} C_VEL
LIN {X 0,Y 559.147,Z 133.838,A -85,B 0,C 180,E1 -3026.424,E2 -3026.424} C_VEL
LIN {X 0,Y 559.148,Z 133.832,A -85,B 0,C 180,E1 -3028.98,E2 -3028.98} C_VEL
LIN {X 0,Y 559.106,Z 133.835,A -85,B 0,C 180,E1 -3031.632,E2 -3031.632} C_VEL
LIN {X 0,Y 559.157,Z 133.832,A -85,B 0,C 180,E1 -3033.902,E2 -3033.902} C_VEL
LIN {X 0,Y 559.114,Z 133.834,A -85,B 0,C 180,E1 -3037.066,E2 -3037.066} C_VEL
LIN {X 0,Y 559.152,Z 133.829,A -85,B 0,C 180,E1 -3039.394,E2 -3039.394} C_VEL
LIN {X 0,Y 559.12,Z 133.837,A -85,B 0,C 180,E1 -3041.685,E2 -3041.685} C_VEL
LIN {X 0,Y 559.134,Z 133.833,A -85,B 0,C 180,E1 -3044.695,E2 -3044.695} C_VEL
LIN {X 0,Y 559.152,Z 133.835,A -85,B 0,C 180,E1 -3047.662,E2 -3047.662} C_VEL
LIN {X 0,Y 559.131,Z 133.842,A -85,B 0,C 180,E1 -3049.865,E2 -3049.865} C_VEL
LIN {X 0,Y 559.147,Z 133.838,A -85,B 0,C 180,E1 -3052.053,E2 -3052.053} C_VEL
LIN {X 0,Y 559.239,Z 133.82,A -85,B 0,C 180,E1 -3054.953,E2 -3054.953} C_VEL
LIN {X 0,Y 559.254,Z 133.825,A -85,B 0,C 180,E1 -3057.84,E2 -3057.84} C_VEL
LIN {X 0,Y 559.259,Z 133.822,A -85,B 0,C 180,E1 -3060,E2 -3060} C_VEL
LIN {X 0,Y 559.224,Z 133.823,A -85,B 0,C 180,E1 -3062.882,E2 -3062.882} C_VEL
LIN {X 0,Y 559.221,Z 133.828,A -85,B 0,C 180,E1 -3065.77,E2 -3065.77} C_VEL
LIN {X 0,Y 559.208,Z 133.857,A -85,B 0,C 180,E1 -3068.265,E2 -3068.265} C_VEL
LIN {X 0,Y 559.46,Z 141.542,A -85,B 0,C 180,E1 -3069.582,E2 -3069.582} C_VEL
LIN {X 0,Y 559.348,Z 157.53,A -85,B 0,C 180,E1 -3072.334,E2 -3072.334} C_VEL
LIN {X 0,Y 559.231,Z 166.235,A -85,B 0,C 180,E1 -3073.861,E2 -3073.861} C_VEL
LIN {X 0,Y 560.351,Z 173.493,A -85,B 0,C 180,E1 -3073.995,E2 -3073.995} C_VEL
LIN {X 0,Y 560.026,Z 271.994,A -85,B 0,C 180,E1 -3075.28,E2 -3075.28} C_VEL
LIN {X 0,Y 559.917,Z 284.702,A -85,B 0,C 180,E1 -3075.563,E2 -3075.563} C_VEL
LIN {X 0,Y 559.881,Z 286.741,A -85,B 0,C 180,E1 -3075.627,E2 -3075.627} C_VEL
LIN {X 0,Y 559.02,Z 292.481,A -85,B 0,C 180,E1 -3075.797,E2 -3075.797} C_VEL
LIN {X 0,Y 556.147,Z 301.714,A -85,B 0,C 180,E1 -3076.11,E2 -3076.11} C_VEL
LIN {X 0,Y 553.284,Z 310.262,A -85,B 0,C 180,E1 -3076.482,E2 -3076.482} C_VEL
LIN {X 0,Y 552.592,Z 315.252,A -85,B 0,C 180,E1 -3076.767,E2 -3076.767} C_VEL
LIN {X 0,Y 552.38,Z 326.432,A -85,B 0,C 180,E1 -3077.54,E2 -3077.54} C_VEL
LIN {X 0,Y 552.2,Z 335.872,A -85,B 0,C 180,E1 -3078.361,E2 -3078.361} C_VEL
LIN {X 0,Y 552.108,Z 343.337,A -85,B 0,C 180,E1 -3079.134,E2 -3079.134} C_VEL
LIN {X 0,Y 551.954,Z 351.246,A -85,B 0,C 180,E1 -3080.108,E2 -3080.108} C_VEL
LIN {X 0,Y 551.856,Z 358.602,A -85,B 0,C 180,E1 -3081.247,E2 -3081.247} C_VEL
LIN {X 0,Y 551.797,Z 363.009,A -85,B 0,C 180,E1 -3082.07,E2 -3082.07} C_VEL
LIN {X 0,Y 551.751,Z 368.211,A -85,B 0,C 180,E1 -3083.258,E2 -3083.258} C_VEL
LIN {X 0,Y 551.735,Z 372.129,A -85,B 0,C 180,E1 -3084.456,E2 -3084.456} C_VEL
LIN {X 0,Y 551.645,Z 374.833,A -85,B 0,C 180,E1 -3085.669,E2 -3085.669} C_VEL
LIN {X 0,Y 551.653,Z 376.476,A -85,B 0,C 180,E1 -3086.9,E2 -3086.9} C_VEL
LIN {X 0,Y 551.667,Z 376.989,A -85,B 0,C 180,E1 -3088.123,E2 -3088.123} C_VEL
LIN {X 0,Y 551.652,Z 376.69,A -85,B 0,C 180,E1 -3088.955,E2 -3088.955} C_VEL
LIN {X 0,Y 551.694,Z 375.611,A -85,B 0,C 180,E1 -3089.974,E2 -3089.974} C_VEL
LIN {X 0,Y 551.737,Z 372.682,A -85,B 0,C 180,E1 -3091.411,E2 -3091.411} C_VEL
LIN {X 0,Y 551.725,Z 368.412,A -85,B 0,C 180,E1 -3092.783,E2 -3092.783} C_VEL
LIN {X 0,Y 551.794,Z 362.696,A -85,B 0,C 180,E1 -3094.085,E2 -3094.085} C_VEL
LIN {X 0,Y 551.87,Z 356.585,A -85,B 0,C 180,E1 -3095.19,E2 -3095.19} C_VEL
LIN {X 0,Y 551.991,Z 348.753,A -85,B 0,C 180,E1 -3096.303,E2 -3096.303} C_VEL
LIN {X 0,Y 552.136,Z 340.072,A -85,B 0,C 180,E1 -3097.316,E2 -3097.316} C_VEL
LIN {X 0,Y 552.284,Z 330.565,A -85,B 0,C 180,E1 -3098.208,E2 -3098.208} C_VEL
LIN {X 0,Y 552.456,Z 320.805,A -85,B 0,C 180,E1 -3098.959,E2 -3098.959} C_VEL
LIN {X 0,Y 552.672,Z 309.573,A -85,B 0,C 180,E1 -3099.659,E2 -3099.659} C_VEL
LIN {X 0,Y 552.87,Z 298.8,A -85,B 0,C 180,E1 -3100.176,E2 -3100.176} C_VEL
LIN {X 0,Y 552.985,Z 286.917,A -85,B 0,C 180,E1 -3100.614,E2 -3100.614} C_VEL
LIN {X 0,Y 553.093,Z 273.125,A -85,B 0,C 180,E1 -3100.95,E2 -3100.95} C_VEL
LIN {X 0,Y 553.376,Z 172.829,A -85,B 0,C 180,E1 -3102.287,E2 -3102.287} C_VEL
LIN {X 0,Y 552.25,Z 166.373,A -85,B 0,C 180,E1 -3102.415,E2 -3102.415} C_VEL
LIN {X 0,Y 552.503,Z 148.684,A -85,B 0,C 180,E1 -3105.603,E2 -3105.603} C_VEL
LIN {X 0,Y 552.542,Z 137.632,A -85,B 0,C 180,E1 -3107.613,E2 -3107.613} C_VEL
LIN {X 0,Y 552.141,Z 134.711,A -85,B 0,C 180,E1 -3108.189,E2 -3108.189} C_VEL
LIN {X 0,Y 552.115,Z 134.707,A -85,B 0,C 180,E1 -3111.41,E2 -3111.41} C_VEL
LIN {X 0,Y 552.075,Z 134.715,A -85,B 0,C 180,E1 -3114.155,E2 -3114.155} C_VEL
LIN {X 0,Y 552.112,Z 134.707,A -85,B 0,C 180,E1 -3117.155,E2 -3117.155} C_VEL
LIN {X 0,Y 552.075,Z 134.713,A -85,B 0,C 180,E1 -3119.958,E2 -3119.958} C_VEL
LIN {X 0,Y 552.083,Z 134.711,A -85,B 0,C 180,E1 -3123.013,E2 -3123.013} C_VEL
LIN {X 0,Y 552.073,Z 134.715,A -85,B 0,C 180,E1 -3125.96,E2 -3125.96} C_VEL
LIN {X 0,Y 552.075,Z 134.711,A -85,B 0,C 180,E1 -3129.117,E2 -3129.117} C_VEL
LIN {X 0,Y 552.069,Z 134.712,A -85,B 0,C 180,E1 -3131.442,E2 -3131.442} C_VEL
LIN {X 0,Y 552.09,Z 134.713,A -85,B 0,C 180,E1 -3134.494,E2 -3134.494} C_VEL
LIN {X 0,Y 552.103,Z 134.708,A -85,B 0,C 180,E1 -3136.754,E2 -3136.754} C_VEL
LIN {X 0,Y 552.088,Z 134.714,A -85,B 0,C 180,E1 -3139.733,E2 -3139.733} C_VEL
LIN {X 0,Y 552.113,Z 134.715,A -85,B 0,C 180,E1 -3141.95,E2 -3141.95} C_VEL
LIN {X 0,Y 552.207,Z 134.694,A -85,B 0,C 180,E1 -3144.888,E2 -3144.888} C_VEL
LIN {X 0,Y 552.223,Z 134.701,A -85,B 0,C 180,E1 -3147.811,E2 -3147.811} C_VEL
LIN {X 0,Y 552.226,Z 134.698,A -85,B 0,C 180,E1 -3149.999,E2 -3149.999} C_VEL
LIN {X 0,Y 552.178,Z 134.698,A -85,B 0,C 180,E1 -3152.918,E2 -3152.918} C_VEL
LIN {X 0,Y 552.177,Z 134.705,A -85,B 0,C 180,E1 -3155.843,E2 -3155.843} C_VEL
LIN {X 0,Y 552.127,Z 134.704,A -85,B 0,C 180,E1 -3158.786,E2 -3158.786} C_VEL
LIN {X 0,Y 552.1,Z 134.714,A -85,B 0,C 180,E1 -3161.751,E2 -3161.751} C_VEL
LIN {X 0,Y 552.122,Z 134.705,A -85,B 0,C 180,E1 -3164.748,E2 -3164.748} C_VEL
LIN {X 0,Y 552.077,Z 134.715,A -85,B 0,C 180,E1 -3167.789,E2 -3167.789} C_VEL
LIN {X 0,Y 552.094,Z 134.709,A -85,B 0,C 180,E1 -3170.102,E2 -3170.102} C_VEL
LIN {X 0,Y 552.043,Z 134.715,A -85,B 0,C 180,E1 -3172.452,E2 -3172.452} C_VEL
LIN {X 0,Y 552.082,Z 134.719,A -85,B 0,C 180,E1 -3175.333,E2 -3175.333} C_VEL
LIN {X 0,Y 552.049,Z 134.714,A -85,B 0,C 180,E1 -3178.101,E2 -3178.101} C_VEL
LIN {X 0,Y 552.068,Z 134.713,A -85,B 0,C 180,E1 -3180.61,E2 -3180.61} C_VEL
LIN {X 0,Y 552.102,Z 134.716,A -85,B 0,C 180,E1 -3183.186,E2 -3183.186} C_VEL
LIN {X 0,Y 552.066,Z 134.712,A -85,B 0,C 180,E1 -3185.844,E2 -3185.844} C_VEL
LIN {X 0,Y 552.11,Z 134.71,A -85,B 0,C 180,E1 -3188.589,E2 -3188.589} C_VEL
LIN {X 0,Y 552.057,Z 134.715,A -85,B 0,C 180,E1 -3191.451,E2 -3191.451} C_VEL
LIN {X 0,Y 552.071,Z 134.715,A -85,B 0,C 180,E1 -3194.529,E2 -3194.529} C_VEL
LIN {X 0,Y 552.078,Z 134.711,A -85,B 0,C 180,E1 -3197.589,E2 -3197.589} C_VEL
LIN {X 0,Y 552.117,Z 134.71,A -85,B 0,C 180,E1 -3200.471,E2 -3200.471} C_VEL
LIN {X 0,Y 552.092,Z 134.71,A -85,B 0,C 180,E1 -3203.318,E2 -3203.318} C_VEL
LIN {X 0,Y 552.09,Z 134.71,A -85,B 0,C 180,E1 -3205.936,E2 -3205.936} C_VEL
LIN {X 0,Y 552.098,Z 134.717,A -85,B 0,C 180,E1 -3208.539,E2 -3208.539} C_VEL
LIN {X 0,Y 552.065,Z 134.712,A -85,B 0,C 180,E1 -3211.448,E2 -3211.448} C_VEL
LIN {X 0,Y 552.075,Z 134.718,A -85,B 0,C 180,E1 -3214.353,E2 -3214.353} C_VEL
LIN {X 0,Y 552.044,Z 134.719,A -85,B 0,C 180,E1 -3216.755,E2 -3216.755} C_VEL
LIN {X 0,Y 552.088,Z 134.71,A -85,B 0,C 180,E1 -3219.118,E2 -3219.118} C_VEL
LIN {X 0,Y 552.069,Z 134.711,A -85,B 0,C 180,E1 -3221.442,E2 -3221.442} C_VEL
LIN {X 0,Y 552.078,Z 134.716,A -85,B 0,C 180,E1 -3224.494,E2 -3224.494} C_VEL
LIN {X 0,Y 552.098,Z 134.709,A -85,B 0,C 180,E1 -3227.502,E2 -3227.502} C_VEL
LIN {X 0,Y 552.078,Z 134.714,A -85,B 0,C 180,E1 -3229.734,E2 -3229.734} C_VEL
LIN {X 0,Y 552.101,Z 134.715,A -85,B 0,C 180,E1 -3231.95,E2 -3231.95} C_VEL
LIN {X 0,Y 552.197,Z 134.696,A -85,B 0,C 180,E1 -3234.888,E2 -3234.888} C_VEL
LIN {X 0,Y 552.213,Z 134.7,A -85,B 0,C 180,E1 -3237.812,E2 -3237.812} C_VEL
LIN {X 0,Y 552.215,Z 134.702,A -85,B 0,C 180,E1 -3240,E2 -3240} C_VEL
LIN {X 0,Y 552.166,Z 134.699,A -85,B 0,C 180,E1 -3242.918,E2 -3242.918} C_VEL
LIN {X 0,Y 552.168,Z 134.709,A -85,B 0,C 180,E1 -3245.844,E2 -3245.844} C_VEL
LIN {X 0,Y 552.115,Z 134.706,A -85,B 0,C 180,E1 -3248.786,E2 -3248.786} C_VEL
LIN {X 0,Y 552.091,Z 134.718,A -85,B 0,C 180,E1 -3251.752,E2 -3251.752} C_VEL
LIN {X 0,Y 552.111,Z 134.706,A -85,B 0,C 180,E1 -3254.749,E2 -3254.749} C_VEL
LIN {X 0,Y 552.065,Z 134.718,A -85,B 0,C 180,E1 -3257.79,E2 -3257.79} C_VEL
LIN {X 0,Y 552.083,Z 134.711,A -85,B 0,C 180,E1 -3260.103,E2 -3260.103} C_VEL
LIN {X 0,Y 552.033,Z 134.716,A -85,B 0,C 180,E1 -3262.453,E2 -3262.453} C_VEL
LIN {X 0,Y 552.072,Z 134.719,A -85,B 0,C 180,E1 -3265.334,E2 -3265.334} C_VEL
LIN {X 0,Y 552.04,Z 134.716,A -85,B 0,C 180,E1 -3268.102,E2 -3268.102} C_VEL
LIN {X 0,Y 552.06,Z 134.713,A -85,B 0,C 180,E1 -3270.612,E2 -3270.612} C_VEL
LIN {X 0,Y 552.095,Z 134.717,A -85,B 0,C 180,E1 -3273.187,E2 -3273.187} C_VEL
LIN {X 0,Y 552.059,Z 134.714,A -85,B 0,C 180,E1 -3275.846,E2 -3275.846} C_VEL
LIN {X 0,Y 552.102,Z 134.709,A -85,B 0,C 180,E1 -3278.59,E2 -3278.59} C_VEL
LIN {X 0,Y 552.055,Z 134.717,A -85,B 0,C 180,E1 -3281.452,E2 -3281.452} C_VEL
LIN {X 0,Y 552.068,Z 134.714,A -85,B 0,C 180,E1 -3284.53,E2 -3284.53} C_VEL
LIN {X 0,Y 552.074,Z 134.712,A -85,B 0,C 180,E1 -3287.591,E2 -3287.591} C_VEL
LIN {X 0,Y 552.087,Z 134.713,A -85,B 0,C 180,E1 -3290.47,E2 -3290.47} C_VEL
LIN {X 0,Y 552.048,Z 134.717,A -85,B 0,C 180,E1 -3293.326,E2 -3293.326} C_VEL
LIN {X 0,Y 552.09,Z 134.709,A -85,B 0,C 180,E1 -3295.937,E2 -3295.937} C_VEL
LIN {X 0,Y 552.076,Z 134.717,A -85,B 0,C 180,E1 -3298.539,E2 -3298.539} C_VEL
LIN {X 0,Y 552.067,Z 134.713,A -85,B 0,C 180,E1 -3301.449,E2 -3301.449} C_VEL
LIN {X 0,Y 552.071,Z 134.719,A -85,B 0,C 180,E1 -3304.354,E2 -3304.354} C_VEL
LIN {X 0,Y 552.08,Z 134.779,A -85,B 0,C 180,E1 -3306.517,E2 -3306.517} C_VEL
LIN {X 0,Y 553.077,Z 141.413,A -85,B 0,C 180,E1 -3307.592,E2 -3307.592} C_VEL
LIN {X 0,Y 552.846,Z 158.286,A -85,B 0,C 180,E1 -3310.173,E2 -3310.173} C_VEL
LIN {X 0,Y 552.544,Z 176.981,A -85,B 0,C 180,E1 -3312.99,E2 -3312.99} C_VEL
LIN {X 0,Y 552.351,Z 194.682,A -85,B 0,C 180,E1 -3315.628,E2 -3315.628} C_VEL
LIN {X 0,Y 553.38,Z 202.226,A -85,B 0,C 180,E1 -3315.764,E2 -3315.764} C_VEL
LIN {X 0,Y 553.105,Z 302.391,A -85,B 0,C 180,E1 -3317.083,E2 -3317.083} C_VEL
LIN {X 0,Y 552.97,Z 315.827,A -85,B 0,C 180,E1 -3317.406,E2 -3317.406} C_VEL
LIN {X 0,Y 552.802,Z 329.204,A -85,B 0,C 180,E1 -3317.892,E2 -3317.892} C_VEL
LIN {X 0,Y 552.643,Z 340.868,A -85,B 0,C 180,E1 -3318.473,E2 -3318.473} C_VEL
LIN {X 0,Y 552.456,Z 352.057,A -85,B 0,C 180,E1 -3319.186,E2 -3319.186} C_VEL
LIN {X 0,Y 552.273,Z 362.529,A -85,B 0,C 180,E1 -3320.016,E2 -3320.016} C_VEL
LIN {X 0,Y 552.125,Z 371.086,A -85,B 0,C 180,E1 -3320.845,E2 -3320.845} C_VEL
LIN {X 0,Y 552.012,Z 378.966,A -85,B 0,C 180,E1 -3321.766,E2 -3321.766} C_VEL
LIN {X 0,Y 551.888,Z 386.625,A -85,B 0,C 180,E1 -3322.868,E2 -3322.868} C_VEL
LIN {X 0,Y 551.867,Z 393.682,A -85,B 0,C 180,E1 -3324.153,E2 -3324.153} C_VEL
LIN {X 0,Y 551.725,Z 398.375,A -85,B 0,C 180,E1 -3325.251,E2 -3325.251} C_VEL
LIN {X 0,Y 551.75,Z 401.96,A -85,B 0,C 180,E1 -3326.349,E2 -3326.349} C_VEL
LIN {X 0,Y 551.723,Z 403.808,A -85,B 0,C 180,E1 -3327.08,E2 -3327.08} C_VEL
LIN {X 0,Y 551.645,Z 406.182,A -85,B 0,C 180,E1 -3328.541,E2 -3328.541} C_VEL
LIN {X 0,Y 551.64,Z 407,A -85,B 0,C 180,E1 -3330.001,E2 -3330.001} C_VEL
LIN {X 0,Y 551.645,Z 406.183,A -85,B 0,C 180,E1 -3331.461,E2 -3331.461} C_VEL
LIN {X 0,Y 551.723,Z 403.809,A -85,B 0,C 180,E1 -3332.921,E2 -3332.921} C_VEL
LIN {X 0,Y 551.764,Z 400.893,A -85,B 0,C 180,E1 -3334.018,E2 -3334.018} C_VEL
LIN {X 0,Y 551.724,Z 396.946,A -85,B 0,C 180,E1 -3335.116,E2 -3335.116} C_VEL
LIN {X 0,Y 551.803,Z 391.186,A -85,B 0,C 180,E1 -3336.342,E2 -3336.342} C_VEL
LIN {X 0,Y 551.927,Z 384.231,A -85,B 0,C 180,E1 -3337.5,E2 -3337.5} C_VEL
LIN {X 0,Y 552.083,Z 375.982,A -85,B 0,C 180,E1 -3338.603,E2 -3338.603} C_VEL
LIN {X 0,Y 552.201,Z 367.475,A -85,B 0,C 180,E1 -3339.524,E2 -3339.524} C_VEL
LIN {X 0,Y 552.413,Z 356.956,A -85,B 0,C 180,E1 -3340.446,E2 -3340.446} C_VEL
LIN {X 0,Y 552.556,Z 346.072,A -85,B 0,C 180,E1 -3341.215,E2 -3341.215} C_VEL
LIN {X 0,Y 552.753,Z 335.107,A -85,B 0,C 180,E1 -3341.831,E2 -3341.831} C_VEL
LIN {X 0,Y 552.9,Z 323.335,A -85,B 0,C 180,E1 -3342.34,E2 -3342.34} C_VEL
LIN {X 0,Y 553.039,Z 310.671,A -85,B 0,C 180,E1 -3342.733,E2 -3342.733} C_VEL
LIN {X 0,Y 553.157,Z 297.726,A -85,B 0,C 180,E1 -3342.987,E2 -3342.987} C_VEL
LIN {X 0,Y 553.194,Z 200.523,A -85,B 0,C 180,E1 -3344.259,E2 -3344.259} C_VEL
LIN {X 0,Y 552.327,Z 194.489,A -85,B 0,C 180,E1 -3344.377,E2 -3344.377} C_VEL
LIN {X 0,Y 552.521,Z 174.477,A -85,B 0,C 180,E1 -3347.337,E2 -3347.337} C_VEL
LIN {X 0,Y 552.793,Z 157.925,A -85,B 0,C 180,E1 -3349.812,E2 -3349.812} C_VEL
LIN {X 0,Y 552.956,Z 140.598,A -85,B 0,C 180,E1 -3352.415,E2 -3352.415} C_VEL
LIN {X 0,Y 552.065,Z 134.721,A -85,B 0,C 180,E1 -3353.364,E2 -3353.364} C_VEL
LIN {X 0,Y 552.072,Z 134.714,A -85,B 0,C 180,E1 -3356.46,E2 -3356.46} C_VEL
LIN {X 0,Y 552.039,Z 134.722,A -85,B 0,C 180,E1 -3358.933,E2 -3358.933} C_VEL
LIN {X 0,Y 552.095,Z 134.715,A -85,B 0,C 180,E1 -3361.472,E2 -3361.472} C_VEL
LIN {X 0,Y 552.095,Z 134.709,A -85,B 0,C 180,E1 -3364.164,E2 -3364.164} C_VEL
LIN {X 0,Y 552.072,Z 134.717,A -85,B 0,C 180,E1 -3366.75,E2 -3366.75} C_VEL
LIN {X 0,Y 552.11,Z 134.709,A -85,B 0,C 180,E1 -3369.529,E2 -3369.529} C_VEL
LIN {X 0,Y 552.085,Z 134.712,A -85,B 0,C 180,E1 -3372.43,E2 -3372.43} C_VEL
LIN {X 0,Y 552.077,Z 134.711,A -85,B 0,C 180,E1 -3375.56,E2 -3375.56} C_VEL
LIN {X 0,Y 552.061,Z 134.718,A -85,B 0,C 180,E1 -3378.548,E2 -3378.548} C_VEL
LIN {X 0,Y 552.112,Z 134.706,A -85,B 0,C 180,E1 -3381.41,E2 -3381.41} C_VEL
LIN {X 0,Y 552.072,Z 134.714,A -85,B 0,C 180,E1 -3384.155,E2 -3384.155} C_VEL
LIN {X 0,Y 552.109,Z 134.708,A -85,B 0,C 180,E1 -3387.155,E2 -3387.155} C_VEL
LIN {X 0,Y 552.076,Z 134.713,A -85,B 0,C 180,E1 -3389.958,E2 -3389.958} C_VEL
LIN {X 0,Y 552.081,Z 134.711,A -85,B 0,C 180,E1 -3393.013,E2 -3393.013} C_VEL
LIN {X 0,Y 552.081,Z 134.715,A -85,B 0,C 180,E1 -3395.961,E2 -3395.961} C_VEL
LIN {X 0,Y 552.112,Z 134.713,A -85,B 0,C 180,E1 -3398.337,E2 -3398.337} C_VEL
LIN {X 0,Y 552.141,Z 134.705,A -85,B 0,C 180,E1 -3400.674,E2 -3400.674} C_VEL
LIN {X 0,Y 552.073,Z 134.716,A -85,B 0,C 180,E1 -3403.736,E2 -3403.736} C_VEL
LIN {X 0,Y 552.118,Z 134.715,A -85,B 0,C 180,E1 -3406.004,E2 -3406.004} C_VEL
LIN {X 0,Y 552.163,Z 134.701,A -85,B 0,C 180,E1 -3408.994,E2 -3408.994} C_VEL
LIN {X 0,Y 552.115,Z 134.715,A -85,B 0,C 180,E1 -3411.951,E2 -3411.951} C_VEL
LIN {X 0,Y 552.215,Z 134.695,A -85,B 0,C 180,E1 -3414.889,E2 -3414.889} C_VEL
LIN {X 0,Y 552.224,Z 134.701,A -85,B 0,C 180,E1 -3417.812,E2 -3417.812} C_VEL
LIN {X 0,Y 552.228,Z 134.698,A -85,B 0,C 180,E1 -3420,E2 -3420} C_VEL
LIN {X 0,Y 552.193,Z 134.7,A -85,B 0,C 180,E1 -3422.918,E2 -3422.918} C_VEL
LIN {X 0,Y 552.19,Z 134.704,A -85,B 0,C 180,E1 -3425.844,E2 -3425.844} C_VEL
LIN {X 0,Y 552.176,Z 134.899,A -85,B 0,C 180,E1 -3428.233,E2 -3428.233} C_VEL
LIN {X 0,Y 552.441,Z 142.428,A -85,B 0,C 180,E1 -3429.52,E2 -3429.52} C_VEL
LIN {X 0,Y 552.327,Z 159.682,A -85,B 0,C 180,E1 -3432.493,E2 -3432.493} C_VEL
LIN {X 0,Y 552.234,Z 166.469,A -85,B 0,C 180,E1 -3433.688,E2 -3433.688} C_VEL
LIN {X 0,Y 553.47,Z 173.974,A -85,B 0,C 180,E1 -3433.821,E2 -3433.821} C_VEL
LIN {X 0,Y 553.12,Z 273.77,A -85,B 0,C 180,E1 -3435.153,E2 -3435.153} C_VEL
LIN {X 0,Y 552.935,Z 287.084,A -85,B 0,C 180,E1 -3435.481,E2 -3435.481} C_VEL
LIN {X 0,Y 552.841,Z 298.695,A -85,B 0,C 180,E1 -3435.909,E2 -3435.909} C_VEL
LIN {X 0,Y 552.655,Z 311.352,A -85,B 0,C 180,E1 -3436.532,E2 -3436.532} C_VEL
LIN {X 0,Y 552.592,Z 315.252,A -85,B 0,C 180,E1 -3436.767,E2 -3436.767} C_VEL
LIN {X 0,Y 551.903,Z 320.312,A -85,B 0,C 180,E1 -3437.077,E2 -3437.077} C_VEL
LIN {X 0,Y 548.957,Z 328.293,A -85,B 0,C 180,E1 -3437.608,E2 -3437.608} C_VEL
LIN {X 0,Y 545.937,Z 335.768,A -85,B 0,C 180,E1 -3438.213,E2 -3438.213} C_VEL
LIN {X 0,Y 545.14,Z 340.021,A -85,B 0,C 180,E1 -3438.636,E2 -3438.636} C_VEL
LIN {X 0,Y 544.981,Z 348.223,A -85,B 0,C 180,E1 -3439.591,E2 -3439.591} C_VEL
LIN {X 0,Y 544.867,Z 355.253,A -85,B 0,C 180,E1 -3440.579,E2 -3440.579} C_VEL
LIN {X 0,Y 544.727,Z 361.929,A -85,B 0,C 180,E1 -3441.73,E2 -3441.73} C_VEL
LIN {X 0,Y 544.669,Z 366.705,A -85,B 0,C 180,E1 -3442.774,E2 -3442.774} C_VEL
LIN {X 0,Y 544.641,Z 371.02,A -85,B 0,C 180,E1 -3443.983,E2 -3443.983} C_VEL
LIN {X 0,Y 544.574,Z 374.545,A -85,B 0,C 180,E1 -3445.393,E2 -3445.393} C_VEL
LIN {X 0,Y 544.567,Z 375.638,A -85,B 0,C 180,E1 -3446.027,E2 -3446.027} C_VEL
LIN {X 0,Y 544.553,Z 376.767,A -85,B 0,C 180,E1 -3447.061,E2 -3447.061} C_VEL
LIN {X 0,Y 544.583,Z 376.931,A -85,B 0,C 180,E1 -3448.65,E2 -3448.65} C_VEL
LIN {X 0,Y 544.603,Z 375.465,A -85,B 0,C 180,E1 -3450.16,E2 -3450.16} C_VEL
LIN {X 0,Y 544.652,Z 372.442,A -85,B 0,C 180,E1 -3451.609,E2 -3451.609} C_VEL
LIN {X 0,Y 544.653,Z 367.977,A -85,B 0,C 180,E1 -3452.992,E2 -3452.992} C_VEL
LIN {X 0,Y 544.72,Z 363.565,A -85,B 0,C 180,E1 -3454.018,E2 -3454.018} C_VEL
LIN {X 0,Y 544.822,Z 356.873,A -85,B 0,C 180,E1 -3455.258,E2 -3455.258} C_VEL
LIN {X 0,Y 544.963,Z 349.071,A -85,B 0,C 180,E1 -3456.387,E2 -3456.387} C_VEL
LIN {X 0,Y 545.13,Z 340.401,A -85,B 0,C 180,E1 -3457.413,E2 -3457.413} C_VEL
LIN {X 0,Y 545.293,Z 330.723,A -85,B 0,C 180,E1 -3458.335,E2 -3458.335} C_VEL
LIN {X 0,Y 545.47,Z 320.211,A -85,B 0,C 180,E1 -3459.149,E2 -3459.149} C_VEL
LIN {X 0,Y 545.716,Z 308.137,A -85,B 0,C 180,E1 -3459.886,E2 -3459.886} C_VEL
LIN {X 0,Y 545.93,Z 295.925,A -85,B 0,C 180,E1 -3460.454,E2 -3460.454} C_VEL
LIN {X 0,Y 546.074,Z 282.709,A -85,B 0,C 180,E1 -3460.895,E2 -3460.895} C_VEL
LIN {X 0,Y 546.207,Z 270.007,A -85,B 0,C 180,E1 -3461.165,E2 -3461.165} C_VEL
LIN {X 0,Y 546.405,Z 173.22,A -85,B 0,C 180,E1 -3462.468,E2 -3462.468} C_VEL
LIN {X 0,Y 545.256,Z 166.501,A -85,B 0,C 180,E1 -3462.609,E2 -3462.609} C_VEL
LIN {X 0,Y 545.528,Z 149.411,A -85,B 0,C 180,E1 -3465.721,E2 -3465.721} C_VEL
LIN {X 0,Y 545.587,Z 139.217,A -85,B 0,C 180,E1 -3467.589,E2 -3467.589} C_VEL
LIN {X 0,Y 545.091,Z 135.59,A -85,B 0,C 180,E1 -3468.323,E2 -3468.323} C_VEL
LIN {X 0,Y 545.078,Z 135.59,A -85,B 0,C 180,E1 -3470.817,E2 -3470.817} C_VEL
LIN {X 0,Y 545.037,Z 135.589,A -85,B 0,C 180,E1 -3473.619,E2 -3473.619} C_VEL
LIN {X 0,Y 545.051,Z 135.592,A -85,B 0,C 180,E1 -3476.327,E2 -3476.327} C_VEL
LIN {X 0,Y 545.051,Z 135.588,A -85,B 0,C 180,E1 -3478.951,E2 -3478.951} C_VEL
LIN {X 0,Y 545.038,Z 135.587,A -85,B 0,C 180,E1 -3481.503,E2 -3481.503} C_VEL
LIN {X 0,Y 545.041,Z 135.591,A -85,B 0,C 180,E1 -3483.997,E2 -3483.997} C_VEL
LIN {X 0,Y 545.059,Z 135.592,A -85,B 0,C 180,E1 -3486.439,E2 -3486.439} C_VEL
LIN {X 0,Y 545.023,Z 135.591,A -85,B 0,C 180,E1 -3488.834,E2 -3488.834} C_VEL
LIN {X 0,Y 545.031,Z 135.588,A -85,B 0,C 180,E1 -3491.193,E2 -3491.193} C_VEL
LIN {X 0,Y 545.021,Z 135.591,A -85,B 0,C 180,E1 -3493.519,E2 -3493.519} C_VEL
LIN {X 0,Y 545.07,Z 135.588,A -85,B 0,C 180,E1 -3495.819,E2 -3495.819} C_VEL
LIN {X 0,Y 545.077,Z 135.583,A -85,B 0,C 180,E1 -3498.848,E2 -3498.848} C_VEL
LIN {X 0,Y 545.071,Z 135.591,A -85,B 0,C 180,E1 -3501.846,E2 -3501.846} C_VEL
LIN {X 0,Y 545.165,Z 135.572,A -85,B 0,C 180,E1 -3504.822,E2 -3504.822} C_VEL
LIN {X 0,Y 545.194,Z 135.576,A -85,B 0,C 180,E1 -3507.783,E2 -3507.783} C_VEL
LIN {X 0,Y 545.195,Z 135.574,A -85,B 0,C 180,E1 -3509.999,E2 -3509.999} C_VEL
LIN {X 0,Y 545.146,Z 135.574,A -85,B 0,C 180,E1 -3512.955,E2 -3512.955} C_VEL
LIN {X 0,Y 545.125,Z 135.582,A -85,B 0,C 180,E1 -3515.919,E2 -3515.919} C_VEL
LIN {X 0,Y 545.07,Z 135.584,A -85,B 0,C 180,E1 -3518.9,E2 -3518.9} C_VEL
LIN {X 0,Y 545.065,Z 135.588,A -85,B 0,C 180,E1 -3521.905,E2 -3521.905} C_VEL
LIN {X 0,Y 545.078,Z 135.584,A -85,B 0,C 180,E1 -3524.943,E2 -3524.943} C_VEL
LIN {X 0,Y 545.045,Z 135.588,A -85,B 0,C 180,E1 -3528.026,E2 -3528.026} C_VEL
LIN {X 0,Y 545.031,Z 135.588,A -85,B 0,C 180,E1 -3530.374,E2 -3530.374} C_VEL
LIN {X 0,Y 544.989,Z 135.595,A -85,B 0,C 180,E1 -3532.759,E2 -3532.759} C_VEL
LIN {X 0,Y 545.033,Z 135.594,A -85,B 0,C 180,E1 -3535.494,E2 -3535.494} C_VEL
LIN {X 0,Y 545.032,Z 135.589,A -85,B 0,C 180,E1 -3538.495,E2 -3538.495} C_VEL
LIN {X 0,Y 545.043,Z 135.589,A -85,B 0,C 180,E1 -3541.675,E2 -3541.675} C_VEL
LIN {X 0,Y 545.043,Z 135.589,A -85,B 0,C 180,E1 -3544.565,E2 -3544.565} C_VEL
LIN {X 0,Y 545.027,Z 135.594,A -85,B 0,C 180,E1 -3547.304,E2 -3547.304} C_VEL
LIN {X 0,Y 545.054,Z 135.586,A -85,B 0,C 180,E1 -3550.143,E2 -3550.143} C_VEL
LIN {X 0,Y 545.014,Z 135.597,A -85,B 0,C 180,E1 -3553.112,E2 -3553.112} C_VEL
LIN {X 0,Y 545.024,Z 135.59,A -85,B 0,C 180,E1 -3556.228,E2 -3556.228} C_VEL
LIN {X 0,Y 545.007,Z 135.599,A -85,B 0,C 180,E1 -3558.878,E2 -3558.878} C_VEL
LIN {X 0,Y 545.039,Z 135.587,A -85,B 0,C 180,E1 -3561.761,E2 -3561.761} C_VEL
LIN {X 0,Y 545.017,Z 135.597,A -85,B 0,C 180,E1 -3564.53,E2 -3564.53} C_VEL
LIN {X 0,Y 545.055,Z 135.587,A -85,B 0,C 180,E1 -3567.21,E2 -3567.21} C_VEL
LIN {X 0,Y 545.017,Z 135.59,A -85,B 0,C 180,E1 -3569.807,E2 -3569.807} C_VEL
LIN {X 0,Y 545.018,Z 135.594,A -85,B 0,C 180,E1 -3572.84,E2 -3572.84} C_VEL
LIN {X 0,Y 545.011,Z 135.591,A -85,B 0,C 180,E1 -3575.629,E2 -3575.629} C_VEL
LIN {X 0,Y 545.027,Z 135.592,A -85,B 0,C 180,E1 -3578.835,E2 -3578.835} C_VEL
LIN {X 0,Y 545.033,Z 135.588,A -85,B 0,C 180,E1 -3581.194,E2 -3581.194} C_VEL
LIN {X 0,Y 545.014,Z 135.591,A -85,B 0,C 180,E1 -3583.519,E2 -3583.519} C_VEL
LIN {X 0,Y 545.056,Z 135.588,A -85,B 0,C 180,E1 -3585.819,E2 -3585.819} C_VEL
LIN {X 0,Y 545.064,Z 135.585,A -85,B 0,C 180,E1 -3588.848,E2 -3588.848} C_VEL
LIN {X 0,Y 545.058,Z 135.59,A -85,B 0,C 180,E1 -3591.846,E2 -3591.846} C_VEL
LIN {X 0,Y 545.156,Z 135.573,A -85,B 0,C 180,E1 -3594.822,E2 -3594.822} C_VEL
LIN {X 0,Y 545.184,Z 135.575,A -85,B 0,C 180,E1 -3597.783,E2 -3597.783} C_VEL
LIN {X 0,Y 545.183,Z 135.578,A -85,B 0,C 180,E1 -3600,E2 -3600} C_VEL
LIN {X 0,Y 545.134,Z 135.575,A -85,B 0,C 180,E1 -3602.956,E2 -3602.956} C_VEL
LIN {X 0,Y 545.118,Z 135.585,A -85,B 0,C 180,E1 -3605.92,E2 -3605.92} C_VEL
LIN {X 0,Y 545.059,Z 135.585,A -85,B 0,C 180,E1 -3608.901,E2 -3608.901} C_VEL
LIN {X 0,Y 545.056,Z 135.591,A -85,B 0,C 180,E1 -3611.906,E2 -3611.906} C_VEL
LIN {X 0,Y 545.067,Z 135.585,A -85,B 0,C 180,E1 -3614.944,E2 -3614.944} C_VEL
LIN {X 0,Y 545.034,Z 135.591,A -85,B 0,C 180,E1 -3618.027,E2 -3618.027} C_VEL
LIN {X 0,Y 545.021,Z 135.59,A -85,B 0,C 180,E1 -3620.375,E2 -3620.375} C_VEL
LIN {X 0,Y 544.979,Z 135.595,A -85,B 0,C 180,E1 -3622.76,E2 -3622.76} C_VEL
LIN {X 0,Y 545.024,Z 135.597,A -85,B 0,C 180,E1 -3625.495,E2 -3625.495} C_VEL
LIN {X 0,Y 545.023,Z 135.589,A -85,B 0,C 180,E1 -3628.497,E2 -3628.497} C_VEL
LIN {X 0,Y 545.036,Z 135.591,A -85,B 0,C 180,E1 -3631.677,E2 -3631.677} C_VEL
LIN {X 0,Y 545.036,Z 135.589,A -85,B 0,C 180,E1 -3634.566,E2 -3634.566} C_VEL
LIN {X 0,Y 545.011,Z 135.598,A -85,B 0,C 180,E1 -3637.306,E2 -3637.306} C_VEL
LIN {X 0,Y 545.026,Z 135.589,A -85,B 0,C 180,E1 -3640.146,E2 -3640.146} C_VEL
LIN {X 0,Y 545.01,Z 135.599,A -85,B 0,C 180,E1 -3643.113,E2 -3643.113} C_VEL
LIN {X 0,Y 545.019,Z 135.59,A -85,B 0,C 180,E1 -3646.23,E2 -3646.23} C_VEL
LIN {X 0,Y 544.998,Z 135.601,A -85,B 0,C 180,E1 -3648.879,E2 -3648.879} C_VEL
LIN {X 0,Y 545.038,Z 135.587,A -85,B 0,C 180,E1 -3651.762,E2 -3651.762} C_VEL
LIN {X 0,Y 545.014,Z 135.595,A -85,B 0,C 180,E1 -3654.531,E2 -3654.531} C_VEL
LIN {X 0,Y 545.048,Z 135.589,A -85,B 0,C 180,E1 -3657.211,E2 -3657.211} C_VEL
LIN {X 0,Y 545.013,Z 135.591,A -85,B 0,C 180,E1 -3659.808,E2 -3659.808} C_VEL
LIN {X 0,Y 544.994,Z 135.598,A -85,B 0,C 180,E1 -3662.34,E2 -3662.34} C_VEL
LIN {X 0,Y 545.032,Z 135.597,A -85,B 0,C 180,E1 -3664.817,E2 -3664.817} C_VEL
LIN {X 0,Y 545.045,Z 135.716,A -85,B 0,C 180,E1 -3666.366,E2 -3666.366} C_VEL
LIN {X 0,Y 546.119,Z 142.416,A -85,B 0,C 180,E1 -3667.473,E2 -3667.473} C_VEL
LIN {X 0,Y 545.884,Z 159.641,A -85,B 0,C 180,E1 -3670.143,E2 -3670.143} C_VEL
LIN {X 0,Y 545.528,Z 178.09,A -85,B 0,C 180,E1 -3672.958,E2 -3672.958} C_VEL
LIN {X 0,Y 545.324,Z 194.546,A -85,B 0,C 180,E1 -3675.445,E2 -3675.445} C_VEL
LIN {X 0,Y 546.493,Z 202.709,A -85,B 0,C 180,E1 -3675.594,E2 -3675.594} C_VEL
LIN {X 0,Y 546.193,Z 301.752,A -85,B 0,C 180,E1 -3676.916,E2 -3676.916} C_VEL
LIN {X 0,Y 546.052,Z 314.607,A -85,B 0,C 180,E1 -3677.22,E2 -3677.22} C_VEL
LIN {X 0,Y 545.85,Z 327.684,A -85,B 0,C 180,E1 -3677.688,E2 -3677.688} C_VEL
LIN {X 0,Y 545.66,Z 339.487,A -85,B 0,C 180,E1 -3678.262,E2 -3678.262} C_VEL
LIN {X 0,Y 545.491,Z 350.456,A -85,B 0,C 180,E1 -3678.952,E2 -3678.952} C_VEL
LIN {X 0,Y 545.247,Z 361.171,A -85,B 0,C 180,E1 -3679.792,E2 -3679.792} C_VEL
LIN {X 0,Y 545.085,Z 370.822,A -85,B 0,C 180,E1 -3680.726,E2 -3680.726} C_VEL
LIN {X 0,Y 544.946,Z 378.73,A -85,B 0,C 180,E1 -3681.658,E2 -3681.658} C_VEL
LIN {X 0,Y 544.823,Z 386.448,A -85,B 0,C 180,E1 -3682.775,E2 -3682.775} C_VEL
LIN {X 0,Y 544.776,Z 393.556,A -85,B 0,C 180,E1 -3684.077,E2 -3684.077} C_VEL
LIN {X 0,Y 544.628,Z 398.278,A -85,B 0,C 180,E1 -3685.189,E2 -3685.189} C_VEL
LIN {X 0,Y 544.669,Z 401.889,A -85,B 0,C 180,E1 -3686.302,E2 -3686.302} C_VEL
LIN {X 0,Y 544.65,Z 403.75,A -85,B 0,C 180,E1 -3687.042,E2 -3687.042} C_VEL
LIN {X 0,Y 544.546,Z 406.137,A -85,B 0,C 180,E1 -3688.522,E2 -3688.522} C_VEL
LIN {X 0,Y 544.542,Z 406.745,A -85,B 0,C 180,E1 -3689.261,E2 -3689.261} C_VEL
LIN {X 0,Y 544.541,Z 406.96,A -85,B 0,C 180,E1 -3690.001,E2 -3690.001} C_VEL
LIN {X 0,Y 544.546,Z 406.137,A -85,B 0,C 180,E1 -3691.48,E2 -3691.48} C_VEL
LIN {X 0,Y 544.65,Z 403.749,A -85,B 0,C 180,E1 -3692.959,E2 -3692.959} C_VEL
LIN {X 0,Y 544.684,Z 400.813,A -85,B 0,C 180,E1 -3694.07,E2 -3694.07} C_VEL
LIN {X 0,Y 544.654,Z 396.834,A -85,B 0,C 180,E1 -3695.183,E2 -3695.183} C_VEL
LIN {X 0,Y 544.712,Z 391.548,A -85,B 0,C 180,E1 -3696.329,E2 -3696.329} C_VEL
LIN {X 0,Y 544.837,Z 385.258,A -85,B 0,C 180,E1 -3697.412,E2 -3697.412} C_VEL
LIN {X 0,Y 544.988,Z 377.203,A -85,B 0,C 180,E1 -3698.529,E2 -3698.529} C_VEL
LIN {X 0,Y 545.114,Z 368.985,A -85,B 0,C 180,E1 -3699.462,E2 -3699.462} C_VEL
LIN {X 0,Y 545.35,Z 358.957,A -85,B 0,C 180,E1 -3700.395,E2 -3700.395} C_VEL
LIN {X 0,Y 545.531,Z 348.028,A -85,B 0,C 180,E1 -3701.209,E2 -3701.209} C_VEL
LIN {X 0,Y 545.71,Z 336.478,A -85,B 0,C 180,E1 -3701.892,E2 -3701.892} C_VEL
LIN {X 0,Y 545.928,Z 324.114,A -85,B 0,C 180,E1 -3702.453,E2 -3702.453} C_VEL
LIN {X 0,Y 546.083,Z 311.903,A -85,B 0,C 180,E1 -3702.851,E2 -3702.851} C_VEL
LIN {X 0,Y 546.2,Z 299.902,A -85,B 0,C 180,E1 -3703.108,E2 -3703.108} C_VEL
LIN {X 0,Y 546.389,Z 201.807,A -85,B 0,C 180,E1 -3704.419,E2 -3704.419} C_VEL
LIN {X 0,Y 545.297,Z 194.305,A -85,B 0,C 180,E1 -3704.56,E2 -3704.56} C_VEL
LIN {X 0,Y 545.521,Z 174.969,A -85,B 0,C 180,E1 -3707.451,E2 -3707.451} C_VEL
LIN {X 0,Y 545.821,Z 157.533,A -85,B 0,C 180,E1 -3710.093,E2 -3710.093} C_VEL
LIN {X 0,Y 545.985,Z 141.512,A -85,B 0,C 180,E1 -3712.523,E2 -3712.523} C_VEL
LIN {X 0,Y 545.043,Z 135.596,A -85,B 0,C 180,E1 -3713.486,E2 -3713.486} C_VEL
LIN {X 0,Y 545.03,Z 135.593,A -85,B 0,C 180,E1 -3716.004,E2 -3716.004} C_VEL
LIN {X 0,Y 545.019,Z 135.594,A -85,B 0,C 180,E1 -3718.734,E2 -3718.734} C_VEL
LIN {X 0,Y 545.046,Z 135.591,A -85,B 0,C 180,E1 -3721.676,E2 -3721.676} C_VEL
LIN {X 0,Y 545.046,Z 135.589,A -85,B 0,C 180,E1 -3724.566,E2 -3724.566} C_VEL
LIN {X 0,Y 545.02,Z 135.596,A -85,B 0,C 180,E1 -3727.306,E2 -3727.306} C_VEL
LIN {X 0,Y 545.057,Z 135.586,A -85,B 0,C 180,E1 -3730.144,E2 -3730.144} C_VEL
LIN {X 0,Y 545.02,Z 135.595,A -85,B 0,C 180,E1 -3733.113,E2 -3733.113} C_VEL
LIN {X 0,Y 545.03,Z 135.589,A -85,B 0,C 180,E1 -3736.229,E2 -3736.229} C_VEL
LIN {X 0,Y 545.014,Z 135.597,A -85,B 0,C 180,E1 -3738.879,E2 -3738.879} C_VEL
LIN {X 0,Y 545.046,Z 135.586,A -85,B 0,C 180,E1 -3741.762,E2 -3741.762} C_VEL
LIN {X 0,Y 545.026,Z 135.596,A -85,B 0,C 180,E1 -3744.531,E2 -3744.531} C_VEL
LIN {X 0,Y 545.064,Z 135.586,A -85,B 0,C 180,E1 -3747.211,E2 -3747.211} C_VEL
LIN {X 0,Y 545.026,Z 135.59,A -85,B 0,C 180,E1 -3749.808,E2 -3749.808} C_VEL
LIN {X 0,Y 545.027,Z 135.592,A -85,B 0,C 180,E1 -3752.841,E2 -3752.841} C_VEL
LIN {X 0,Y 545.023,Z 135.59,A -85,B 0,C 180,E1 -3755.63,E2 -3755.63} C_VEL
LIN {X 0,Y 545.068,Z 135.592,A -85,B 0,C 180,E1 -3758.181,E2 -3758.181} C_VEL
LIN {X 0,Y 545.106,Z 135.585,A -85,B 0,C 180,E1 -3760.414,E2 -3760.414} C_VEL
LIN {X 0,Y 545.021,Z 135.592,A -85,B 0,C 180,E1 -3763.52,E2 -3763.52} C_VEL
LIN {X 0,Y 545.083,Z 135.589,A -85,B 0,C 180,E1 -3765.82,E2 -3765.82} C_VEL
LIN {X 0,Y 545.119,Z 135.579,A -85,B 0,C 180,E1 -3768.849,E2 -3768.849} C_VEL
LIN {X 0,Y 545.073,Z 135.593,A -85,B 0,C 180,E1 -3771.846,E2 -3771.846} C_VEL
LIN {X 0,Y 545.173,Z 135.572,A -85,B 0,C 180,E1 -3774.823,E2 -3774.823} C_VEL
LIN {X 0,Y 545.195,Z 135.577,A -85,B 0,C 180,E1 -3777.784,E2 -3777.784} C_VEL
LIN {X 0,Y 545.197,Z 135.574,A -85,B 0,C 180,E1 -3780,E2 -3780} C_VEL
LIN {X 0,Y 545.161,Z 135.576,A -85,B 0,C 180,E1 -3782.956,E2 -3782.956} C_VEL
LIN {X 0,Y 545.14,Z 135.582,A -85,B 0,C 180,E1 -3785.92,E2 -3785.92} C_VEL
LIN {X 0,Y 545.163,Z 135.773,A -85,B 0,C 180,E1 -3788.153,E2 -3788.153} C_VEL
LIN {X 0,Y 545.482,Z 142.193,A -85,B 0,C 180,E1 -3789.268,E2 -3789.268} C_VEL
LIN {X 0,Y 545.322,Z 159.65,A -85,B 0,C 180,E1 -3792.278,E2 -3792.278} C_VEL
LIN {X 0,Y 545.229,Z 166.469,A -85,B 0,C 180,E1 -3793.487,E2 -3793.487} C_VEL
LIN {X 0,Y 546.561,Z 174.44,A -85,B 0,C 180,E1 -3793.643,E2 -3793.643} C_VEL
LIN {X 0,Y 546.204,Z 273.888,A -85,B 0,C 180,E1 -3794.993,E2 -3794.993} C_VEL
LIN {X 0,Y 546.02,Z 287.164,A -85,B 0,C 180,E1 -3795.324,E2 -3795.324} C_VEL
LIN {X 0,Y 545.89,Z 299.387,A -85,B 0,C 180,E1 -3795.782,E2 -3795.782} C_VEL
LIN {X 0,Y 545.688,Z 311.077,A -85,B 0,C 180,E1 -3796.364,E2 -3796.364} C_VEL
LIN {X 0,Y 545.465,Z 321.674,A -85,B 0,C 180,E1 -3797.045,E2 -3797.045} C_VEL
LIN {X 0,Y 545.283,Z 332.056,A -85,B 0,C 180,E1 -3797.867,E2 -3797.867} C_VEL
LIN {X 0,Y 545.14,Z 340.021,A -85,B 0,C 180,E1 -3798.636,E2 -3798.636} C_VEL
LIN {X 0,Y 544.361,Z 344.17,A -85,B 0,C 180,E1 -3799.081,E2 -3799.081} C_VEL
LIN {X 0,Y 541.381,Z 350.512,A -85,B 0,C 180,E1 -3799.823,E2 -3799.823} C_VEL
LIN {X 0,Y 538.447,Z 356.25,A -85,B 0,C 180,E1 -3800.619,E2 -3800.619} C_VEL
LIN {X 0,Y 537.738,Z 359.384,A -85,B 0,C 180,E1 -3801.144,E2 -3801.144} C_VEL
LIN {X 0,Y 537.651,Z 365.096,A -85,B 0,C 180,E1 -3802.277,E2 -3802.277} C_VEL
LIN {X 0,Y 537.586,Z 369.627,A -85,B 0,C 180,E1 -3803.43,E2 -3803.43} C_VEL
LIN {X 0,Y 537.514,Z 373.375,A -85,B 0,C 180,E1 -3804.734,E2 -3804.734} C_VEL
LIN {X 0,Y 537.485,Z 375.101,A -85,B 0,C 180,E1 -3805.563,E2 -3805.563} C_VEL
LIN {X 0,Y 537.456,Z 376.326,A -85,B 0,C 180,E1 -3806.398,E2 -3806.398} C_VEL
LIN {X 0,Y 537.46,Z 377.073,A -85,B 0,C 180,E1 -3807.237,E2 -3807.237} C_VEL
LIN {X 0,Y 537.459,Z 377.308,A -85,B 0,C 180,E1 -3808.083,E2 -3808.083} C_VEL
LIN {X 0,Y 537.487,Z 377.021,A -85,B 0,C 180,E1 -3808.934,E2 -3808.934} C_VEL
LIN {X 0,Y 537.517,Z 375.388,A -85,B 0,C 180,E1 -3810.35,E2 -3810.35} C_VEL
LIN {X 0,Y 537.556,Z 372.242,A -85,B 0,C 180,E1 -3811.808,E2 -3811.808} C_VEL
LIN {X 0,Y 537.58,Z 367.576,A -85,B 0,C 180,E1 -3813.206,E2 -3813.206} C_VEL
LIN {X 0,Y 537.653,Z 363.245,A -85,B 0,C 180,E1 -3814.2,E2 -3814.2} C_VEL
LIN {X 0,Y 537.777,Z 356.141,A -85,B 0,C 180,E1 -3815.494,E2 -3815.494} C_VEL
LIN {X 0,Y 537.908,Z 349.376,A -85,B 0,C 180,E1 -3816.476,E2 -3816.476} C_VEL
LIN {X 0,Y 538.105,Z 341.005,A -85,B 0,C 180,E1 -3817.483,E2 -3817.483} C_VEL
LIN {X 0,Y 538.283,Z 331.313,A -85,B 0,C 180,E1 -3818.428,E2 -3818.428} C_VEL
LIN {X 0,Y 538.484,Z 320.602,A -85,B 0,C 180,E1 -3819.272,E2 -3819.272} C_VEL
LIN {X 0,Y 538.746,Z 308.227,A -85,B 0,C 180,E1 -3820.038,E2 -3820.038} C_VEL
LIN {X 0,Y 538.987,Z 297.067,A -85,B 0,C 180,E1 -3820.567,E2 -3820.567} C_VEL
LIN {X 0,Y 539.155,Z 284.124,A -85,B 0,C 180,E1 -3821.023,E2 -3821.023} C_VEL
LIN {X 0,Y 539.28,Z 271.411,A -85,B 0,C 180,E1 -3821.308,E2 -3821.308} C_VEL
LIN {X 0,Y 539.587,Z 174.361,A -85,B 0,C 180,E1 -3822.639,E2 -3822.639} C_VEL
LIN {X 0,Y 538.261,Z 166.69,A -85,B 0,C 180,E1 -3822.794,E2 -3822.794} C_VEL
LIN {X 0,Y 538.547,Z 148.969,A -85,B 0,C 180,E1 -3826.055,E2 -3826.055} C_VEL
LIN {X 0,Y 538.556,Z 139.916,A -85,B 0,C 180,E1 -3827.739,E2 -3827.739} C_VEL
LIN {X 0,Y 538.054,Z 136.467,A -85,B 0,C 180,E1 -3828.416,E2 -3828.416} C_VEL
LIN {X 0,Y 537.999,Z 136.465,A -85,B 0,C 180,E1 -3831.61,E2 -3831.61} C_VEL
LIN {X 0,Y 537.974,Z 136.471,A -85,B 0,C 180,E1 -3834.093,E2 -3834.093} C_VEL
LIN {X 0,Y 538.037,Z 136.465,A -85,B 0,C 180,E1 -3836.727,E2 -3836.727} C_VEL
LIN {X 0,Y 537.995,Z 136.465,A -85,B 0,C 180,E1 -3839.563,E2 -3839.563} C_VEL
LIN {X 0,Y 538.002,Z 136.469,A -85,B 0,C 180,E1 -3842.661,E2 -3842.661} C_VEL
LIN {X 0,Y 537.978,Z 136.467,A -85,B 0,C 180,E1 -3845.289,E2 -3845.289} C_VEL
LIN {X 0,Y 538,Z 136.47,A -85,B 0,C 180,E1 -3848.048,E2 -3848.048} C_VEL
LIN {X 0,Y 537.989,Z 136.466,A -85,B 0,C 180,E1 -3850.938,E2 -3850.938} C_VEL
LIN {X 0,Y 537.968,Z 136.468,A -85,B 0,C 180,E1 -3853.297,E2 -3853.297} C_VEL
LIN {X 0,Y 538.044,Z 136.461,A -85,B 0,C 180,E1 -3855.63,E2 -3855.63} C_VEL
LIN {X 0,Y 538.029,Z 136.462,A -85,B 0,C 180,E1 -3858.7,E2 -3858.7} C_VEL
LIN {X 0,Y 538.039,Z 136.465,A -85,B 0,C 180,E1 -3861.738,E2 -3861.738} C_VEL
LIN {X 0,Y 538.125,Z 136.449,A -85,B 0,C 180,E1 -3864.754,E2 -3864.754} C_VEL
LIN {X 0,Y 538.165,Z 136.451,A -85,B 0,C 180,E1 -3867.754,E2 -3867.754} C_VEL
LIN {X 0,Y 538.163,Z 136.45,A -85,B 0,C 180,E1 -3869.999,E2 -3869.999} C_VEL
LIN {X 0,Y 538.114,Z 136.45,A -85,B 0,C 180,E1 -3872.994,E2 -3872.994} C_VEL
LIN {X 0,Y 538.078,Z 136.459,A -85,B 0,C 180,E1 -3875.997,E2 -3875.997} C_VEL
LIN {X 0,Y 538.028,Z 136.462,A -85,B 0,C 180,E1 -3879.018,E2 -3879.018} C_VEL
LIN {X 0,Y 538.035,Z 136.462,A -85,B 0,C 180,E1 -3882.063,E2 -3882.063} C_VEL
LIN {X 0,Y 538.038,Z 136.463,A -85,B 0,C 180,E1 -3885.143,E2 -3885.143} C_VEL
LIN {X 0,Y 537.998,Z 136.465,A -85,B 0,C 180,E1 -3888.271,E2 -3888.271} C_VEL
LIN {X 0,Y 537.989,Z 136.466,A -85,B 0,C 180,E1 -3890.653,E2 -3890.653} C_VEL
LIN {X 0,Y 537.976,Z 136.472,A -85,B 0,C 180,E1 -3893.073,E2 -3893.073} C_VEL
LIN {X 0,Y 537.992,Z 136.469,A -85,B 0,C 180,E1 -3895.66,E2 -3895.66} C_VEL
LIN {X 0,Y 537.971,Z 136.468,A -85,B 0,C 180,E1 -3898.053,E2 -3898.053} C_VEL
LIN {X 0,Y 537.987,Z 136.468,A -85,B 0,C 180,E1 -3900.628,E2 -3900.628} C_VEL
LIN {X 0,Y 538.019,Z 136.469,A -85,B 0,C 180,E1 -3903.278,E2 -3903.278} C_VEL
LIN {X 0,Y 537.967,Z 136.468,A -85,B 0,C 180,E1 -3906.006,E2 -3906.006} C_VEL
LIN {X 0,Y 538.006,Z 136.47,A -85,B 0,C 180,E1 -3908.83,E2 -3908.83} C_VEL
LIN {X 0,Y 537.977,Z 136.467,A -85,B 0,C 180,E1 -3911.872,E2 -3911.872} C_VEL
LIN {X 0,Y 537.99,Z 136.475,A -85,B 0,C 180,E1 -3914.863,E2 -3914.863} C_VEL
LIN {X 0,Y 537.968,Z 136.472,A -85,B 0,C 180,E1 -3917.208,E2 -3917.208} C_VEL
LIN {X 0,Y 538.002,Z 136.468,A -85,B 0,C 180,E1 -3920.418,E2 -3920.418} C_VEL
LIN {X 0,Y 538.012,Z 136.467,A -85,B 0,C 180,E1 -3923.066,E2 -3923.066} C_VEL
LIN {X 0,Y 537.991,Z 136.465,A -85,B 0,C 180,E1 -3925.824,E2 -3925.824} C_VEL
LIN {X 0,Y 537.989,Z 136.473,A -85,B 0,C 180,E1 -3928.497,E2 -3928.497} C_VEL
LIN {X 0,Y 537.978,Z 136.469,A -85,B 0,C 180,E1 -3931.095,E2 -3931.095} C_VEL
LIN {X 0,Y 537.978,Z 136.467,A -85,B 0,C 180,E1 -3933.63,E2 -3933.63} C_VEL
LIN {X 0,Y 537.977,Z 136.472,A -85,B 0,C 180,E1 -3936.127,E2 -3936.127} C_VEL
LIN {X 0,Y 537.991,Z 136.472,A -85,B 0,C 180,E1 -3938.544,E2 -3938.544} C_VEL
LIN {X 0,Y 537.998,Z 136.466,A -85,B 0,C 180,E1 -3940.938,E2 -3940.938} C_VEL
LIN {X 0,Y 537.962,Z 136.469,A -85,B 0,C 180,E1 -3943.297,E2 -3943.297} C_VEL
LIN {X 0,Y 538.029,Z 136.462,A -85,B 0,C 180,E1 -3945.629,E2 -3945.629} C_VEL
LIN {X 0,Y 538.016,Z 136.464,A -85,B 0,C 180,E1 -3948.7,E2 -3948.7} C_VEL
LIN {X 0,Y 538.027,Z 136.465,A -85,B 0,C 180,E1 -3951.738,E2 -3951.738} C_VEL
LIN {X 0,Y 538.116,Z 136.45,A -85,B 0,C 180,E1 -3954.754,E2 -3954.754} C_VEL
LIN {X 0,Y 538.155,Z 136.45,A -85,B 0,C 180,E1 -3957.754,E2 -3957.754} C_VEL
LIN {X 0,Y 538.152,Z 136.454,A -85,B 0,C 180,E1 -3960,E2 -3960} C_VEL
LIN {X 0,Y 538.102,Z 136.451,A -85,B 0,C 180,E1 -3962.995,E2 -3962.995} C_VEL
LIN {X 0,Y 538.073,Z 136.462,A -85,B 0,C 180,E1 -3965.998,E2 -3965.998} C_VEL
LIN {X 0,Y 538.017,Z 136.463,A -85,B 0,C 180,E1 -3969.018,E2 -3969.018} C_VEL
LIN {X 0,Y 538.026,Z 136.465,A -85,B 0,C 180,E1 -3972.064,E2 -3972.064} C_VEL
LIN {X 0,Y 538.027,Z 136.463,A -85,B 0,C 180,E1 -3975.144,E2 -3975.144} C_VEL
LIN {X 0,Y 537.987,Z 136.466,A -85,B 0,C 180,E1 -3978.272,E2 -3978.272} C_VEL
LIN {X 0,Y 537.978,Z 136.467,A -85,B 0,C 180,E1 -3980.654,E2 -3980.654} C_VEL
LIN {X 0,Y 537.967,Z 136.472,A -85,B 0,C 180,E1 -3983.074,E2 -3983.074} C_VEL
LIN {X 0,Y 537.983,Z 136.472,A -85,B 0,C 180,E1 -3985.661,E2 -3985.661} C_VEL
LIN {X 0,Y 537.963,Z 136.47,A -85,B 0,C 180,E1 -3988.054,E2 -3988.054} C_VEL
LIN {X 0,Y 537.979,Z 136.468,A -85,B 0,C 180,E1 -3990.629,E2 -3990.629} C_VEL
LIN {X 0,Y 538.013,Z 136.472,A -85,B 0,C 180,E1 -3993.279,E2 -3993.279} C_VEL
LIN {X 0,Y 537.953,Z 136.47,A -85,B 0,C 180,E1 -3996.008,E2 -3996.008} C_VEL
LIN {X 0,Y 537.993,Z 136.47,A -85,B 0,C 180,E1 -3998.832,E2 -3998.832} C_VEL
LIN {X 0,Y 537.974,Z 136.468,A -85,B 0,C 180,E1 -4001.873,E2 -4001.873} C_VEL
LIN {X 0,Y 537.987,Z 136.473,A -85,B 0,C 180,E1 -4004.864,E2 -4004.864} C_VEL
LIN {X 0,Y 537.964,Z 136.474,A -85,B 0,C 180,E1 -4007.21,E2 -4007.21} C_VEL
LIN {X 0,Y 537.981,Z 136.467,A -85,B 0,C 180,E1 -4010.2,E2 -4010.2} C_VEL
LIN {X 0,Y 537.954,Z 136.476,A -85,B 0,C 180,E1 -4013.062,E2 -4013.062} C_VEL
LIN {X 0,Y 537.99,Z 136.465,A -85,B 0,C 180,E1 -4015.826,E2 -4015.826} C_VEL
LIN {X 0,Y 537.985,Z 136.472,A -85,B 0,C 180,E1 -4018.498,E2 -4018.498} C_VEL
LIN {X 0,Y 537.981,Z 136.47,A -85,B 0,C 180,E1 -4021.096,E2 -4021.096} C_VEL
LIN {X 0,Y 537.976,Z 136.469,A -85,B 0,C 180,E1 -4023.631,E2 -4023.631} C_VEL
LIN {X 0,Y 538.001,Z 136.673,A -85,B 0,C 180,E1 -4026.213,E2 -4026.213} C_VEL
LIN {X 0,Y 539.193,Z 143.915,A -85,B 0,C 180,E1 -4027.428,E2 -4027.428} C_VEL
LIN {X 0,Y 538.891,Z 161.43,A -85,B 0,C 180,E1 -4030.18,E2 -4030.18} C_VEL
LIN {X 0,Y 538.541,Z 180.468,A -85,B 0,C 180,E1 -4033.121,E2 -4033.121} C_VEL
LIN {X 0,Y 538.294,Z 194.506,A -85,B 0,C 180,E1 -4035.257,E2 -4035.257} C_VEL
LIN {X 0,Y 539.611,Z 204.309,A -85,B 0,C 180,E1 -4035.432,E2 -4035.432} C_VEL
LIN {X 0,Y 539.275,Z 302.404,A -85,B 0,C 180,E1 -4036.77,E2 -4036.77} C_VEL
LIN {X 0,Y 539.095,Z 315.681,A -85,B 0,C 180,E1 -4037.101,E2 -4037.101} C_VEL
LIN {X 0,Y 538.888,Z 328.423,A -85,B 0,C 180,E1 -4037.574,E2 -4037.574} C_VEL
LIN {X 0,Y 538.658,Z 340.072,A -85,B 0,C 180,E1 -4038.161,E2 -4038.161} C_VEL
LIN {X 0,Y 538.466,Z 351.449,A -85,B 0,C 180,E1 -4038.901,E2 -4038.901} C_VEL
LIN {X 0,Y 538.196,Z 361.963,A -85,B 0,C 180,E1 -4039.752,E2 -4039.752} C_VEL
LIN {X 0,Y 538.046,Z 370.559,A -85,B 0,C 180,E1 -4040.604,E2 -4040.604} C_VEL
LIN {X 0,Y 537.898,Z 378.483,A -85,B 0,C 180,E1 -4041.548,E2 -4041.548} C_VEL
LIN {X 0,Y 537.754,Z 386.218,A -85,B 0,C 180,E1 -4042.68,E2 -4042.68} C_VEL
LIN {X 0,Y 537.684,Z 393.336,A -85,B 0,C 180,E1 -4043.998,E2 -4043.998} C_VEL
LIN {X 0,Y 537.54,Z 398.068,A -85,B 0,C 180,E1 -4045.126,E2 -4045.126} C_VEL
LIN {X 0,Y 537.591,Z 401.687,A -85,B 0,C 180,E1 -4046.253,E2 -4046.253} C_VEL
LIN {X 0,Y 537.551,Z 403.551,A -85,B 0,C 180,E1 -4047.003,E2 -4047.003} C_VEL
LIN {X 0,Y 537.49,Z 404.947,A -85,B 0,C 180,E1 -4047.753,E2 -4047.753} C_VEL
LIN {X 0,Y 537.444,Z 406.551,A -85,B 0,C 180,E1 -4049.251,E2 -4049.251} C_VEL
LIN {X 0,Y 537.444,Z 406.766,A -85,B 0,C 180,E1 -4050.001,E2 -4050.001} C_VEL
LIN {X 0,Y 537.451,Z 405.94,A -85,B 0,C 180,E1 -4051.499,E2 -4051.499} C_VEL
LIN {X 0,Y 537.49,Z 404.943,A -85,B 0,C 180,E1 -4052.249,E2 -4052.249} C_VEL
LIN {X 0,Y 537.551,Z 403.543,A -85,B 0,C 180,E1 -4052.998,E2 -4052.998} C_VEL
LIN {X 0,Y 537.603,Z 400.599,A -85,B 0,C 180,E1 -4054.124,E2 -4054.124} C_VEL
LIN {X 0,Y 537.587,Z 396.61,A -85,B 0,C 180,E1 -4055.251,E2 -4055.251} C_VEL
LIN {X 0,Y 537.618,Z 391.819,A -85,B 0,C 180,E1 -4056.31,E2 -4056.31} C_VEL
LIN {X 0,Y 537.754,Z 385.001,A -85,B 0,C 180,E1 -4057.51,E2 -4057.51} C_VEL
LIN {X 0,Y 537.91,Z 376.928,A -85,B 0,C 180,E1 -4058.642,E2 -4058.642} C_VEL
LIN {X 0,Y 538.069,Z 368.691,A -85,B 0,C 180,E1 -4059.587,E2 -4059.587} C_VEL
LIN {X 0,Y 538.322,Z 358.632,A -85,B 0,C 180,E1 -4060.532,E2 -4060.532} C_VEL
LIN {X 0,Y 538.515,Z 348.676,A -85,B 0,C 180,E1 -4061.29,E2 -4061.29} C_VEL
LIN {X 0,Y 538.704,Z 337.672,A -85,B 0,C 180,E1 -4061.963,E2 -4061.963} C_VEL
LIN {X 0,Y 538.941,Z 324.799,A -85,B 0,C 180,E1 -4062.569,E2 -4062.569} C_VEL
LIN {X 0,Y 539.139,Z 312.217,A -85,B 0,C 180,E1 -4062.995,E2 -4062.995} C_VEL
LIN {X 0,Y 539.279,Z 299.064,A -85,B 0,C 180,E1 -4063.28,E2 -4063.28} C_VEL
LIN {X 0,Y 539.492,Z 202.248,A -85,B 0,C 180,E1 -4064.598,E2 -4064.598} C_VEL
LIN {X 0,Y 538.246,Z 194.032,A -85,B 0,C 180,E1 -4064.762,E2 -4064.762} C_VEL
LIN {X 0,Y 538.515,Z 176.117,A -85,B 0,C 180,E1 -4067.468,E2 -4067.468} C_VEL
LIN {X 0,Y 538.787,Z 160.722,A -85,B 0,C 180,E1 -4069.825,E2 -4069.825} C_VEL
LIN {X 0,Y 539.011,Z 142.578,A -85,B 0,C 180,E1 -4072.622,E2 -4072.622} C_VEL
LIN {X 0,Y 537.993,Z 136.474,A -85,B 0,C 180,E1 -4073.627,E2 -4073.627} C_VEL
LIN {X 0,Y 537.978,Z 136.471,A -85,B 0,C 180,E1 -4076.371,E2 -4076.371} C_VEL
LIN {X 0,Y 537.976,Z 136.474,A -85,B 0,C 180,E1 -4078.922,E2 -4078.922} C_VEL
LIN {X 0,Y 537.998,Z 136.467,A -85,B 0,C 180,E1 -4081.885,E2 -4081.885} C_VEL
LIN {X 0,Y 537.996,Z 136.468,A -85,B 0,C 180,E1 -4084.615,E2 -4084.615} C_VEL
LIN {X 0,Y 537.984,Z 136.467,A -85,B 0,C 180,E1 -4087.879,E2 -4087.879} C_VEL
LIN {X 0,Y 538,Z 136.471,A -85,B 0,C 180,E1 -4090.781,E2 -4090.781} C_VEL
LIN {X 0,Y 538.003,Z 136.464,A -85,B 0,C 180,E1 -4094.071,E2 -4094.071} C_VEL
LIN {X 0,Y 537.971,Z 136.473,A -85,B 0,C 180,E1 -4097.019,E2 -4097.019} C_VEL
LIN {X 0,Y 538.003,Z 136.466,A -85,B 0,C 180,E1 -4100.201,E2 -4100.201} C_VEL
LIN {X 0,Y 538.02,Z 136.464,A -85,B 0,C 180,E1 -4103.067,E2 -4103.067} C_VEL
LIN {X 0,Y 538,Z 136.466,A -85,B 0,C 180,E1 -4105.825,E2 -4105.825} C_VEL
LIN {X 0,Y 537.997,Z 136.473,A -85,B 0,C 180,E1 -4108.498,E2 -4108.498} C_VEL
LIN {X 0,Y 537.987,Z 136.466,A -85,B 0,C 180,E1 -4111.096,E2 -4111.096} C_VEL
LIN {X 0,Y 537.987,Z 136.467,A -85,B 0,C 180,E1 -4113.63,E2 -4113.63} C_VEL
LIN {X 0,Y 538.01,Z 136.47,A -85,B 0,C 180,E1 -4116.123,E2 -4116.123} C_VEL
LIN {X 0,Y 538.015,Z 136.466,A -85,B 0,C 180,E1 -4118.546,E2 -4118.546} C_VEL
LIN {X 0,Y 538.009,Z 136.464,A -85,B 0,C 180,E1 -4120.939,E2 -4120.939} C_VEL
LIN {X 0,Y 537.969,Z 136.469,A -85,B 0,C 180,E1 -4123.297,E2 -4123.297} C_VEL
LIN {X 0,Y 538.056,Z 136.462,A -85,B 0,C 180,E1 -4125.631,E2 -4125.631} C_VEL
LIN {X 0,Y 538.08,Z 136.456,A -85,B 0,C 180,E1 -4128.702,E2 -4128.702} C_VEL
LIN {X 0,Y 538.044,Z 136.468,A -85,B 0,C 180,E1 -4131.739,E2 -4131.739} C_VEL
LIN {X 0,Y 538.132,Z 136.449,A -85,B 0,C 180,E1 -4134.755,E2 -4134.755} C_VEL
LIN {X 0,Y 538.167,Z 136.453,A -85,B 0,C 180,E1 -4137.755,E2 -4137.755} C_VEL
LIN {X 0,Y 538.166,Z 136.45,A -85,B 0,C 180,E1 -4140,E2 -4140} C_VEL
LIN {X 0,Y 538.129,Z 136.453,A -85,B 0,C 180,E1 -4142.995,E2 -4142.995} C_VEL
LIN {X 0,Y 538.096,Z 136.459,A -85,B 0,C 180,E1 -4145.998,E2 -4145.998} C_VEL
LIN {X 0,Y 538.107,Z 136.579,A -85,B 0,C 180,E1 -4148.048,E2 -4148.048} C_VEL
LIN {X 0,Y 538.43,Z 141.005,A -85,B 0,C 180,E1 -4148.823,E2 -4148.823} C_VEL
LIN {X 0,Y 538.346,Z 155.272,A -85,B 0,C 180,E1 -4151.293,E2 -4151.293} C_VEL
LIN {X 0,Y 538.261,Z 166.736,A -85,B 0,C 180,E1 -4153.305,E2 -4153.305} C_VEL
LIN {X 0,Y 539.663,Z 174.888,A -85,B 0,C 180,E1 -4153.461,E2 -4153.461} C_VEL
LIN {X 0,Y 539.268,Z 273.426,A -85,B 0,C 180,E1 -4154.819,E2 -4154.819} C_VEL
LIN {X 0,Y 539.108,Z 287.128,A -85,B 0,C 180,E1 -4155.161,E2 -4155.161} C_VEL
LIN {X 0,Y 538.964,Z 299.488,A -85,B 0,C 180,E1 -4155.626,E2 -4155.626} C_VEL
LIN {X 0,Y 538.717,Z 310.806,A -85,B 0,C 180,E1 -4156.192,E2 -4156.192} C_VEL
LIN {X 0,Y 538.502,Z 321.494,A -85,B 0,C 180,E1 -4156.881,E2 -4156.881} C_VEL
LIN {X 0,Y 538.279,Z 332.406,A -85,B 0,C 180,E1 -4157.756,E2 -4157.756} C_VEL
LIN {X 0,Y 538.077,Z 341.547,A -85,B 0,C 180,E1 -4158.663,E2 -4158.663} C_VEL
LIN {X 0,Y 537.91,Z 349.593,A -85,B 0,C 180,E1 -4159.638,E2 -4159.638} C_VEL
LIN {X 0,Y 537.781,Z 356.595,A -85,B 0,C 180,E1 -4160.662,E2 -4160.662} C_VEL
LIN {X 0,Y 537.738,Z 359.384,A -85,B 0,C 180,E1 -4161.144,E2 -4161.144} C_VEL
LIN {X 0,Y 537.019,Z 362.345,A -85,B 0,C 180,E1 -4161.686,E2 -4161.686} C_VEL
LIN {X 0,Y 534.059,Z 366.674,A -85,B 0,C 180,E1 -4162.588,E2 -4162.588} C_VEL
LIN {X 0,Y 531.133,Z 370.316,A -85,B 0,C 180,E1 -4163.532,E2 -4163.532} C_VEL
LIN {X 0,Y 530.477,Z 372.163,A -85,B 0,C 180,E1 -4164.134,E2 -4164.134} C_VEL
LIN {X 0,Y 530.402,Z 374.491,A -85,B 0,C 180,E1 -4165.088,E2 -4165.088} C_VEL
LIN {X 0,Y 530.371,Z 375.957,A -85,B 0,C 180,E1 -4165.931,E2 -4165.931} C_VEL
LIN {X 0,Y 530.374,Z 377.342,A -85,B 0,C 180,E1 -4167.399,E2 -4167.399} C_VEL
LIN {X 0,Y 530.4,Z 377.167,A -85,B 0,C 180,E1 -4169.01,E2 -4169.01} C_VEL
LIN {X 0,Y 530.443,Z 375.309,A -85,B 0,C 180,E1 -4170.547,E2 -4170.547} C_VEL
LIN {X 0,Y 530.468,Z 371.981,A -85,B 0,C 180,E1 -4172.014,E2 -4172.014} C_VEL
LIN {X 0,Y 530.512,Z 367.177,A -85,B 0,C 180,E1 -4173.425,E2 -4173.425} C_VEL
LIN {X 0,Y 530.62,Z 360.84,A -85,B 0,C 180,E1 -4174.796,E2 -4174.796} C_VEL
LIN {X 0,Y 530.768,Z 354.414,A -85,B 0,C 180,E1 -4175.884,E2 -4175.884} C_VEL
LIN {X 0,Y 530.948,Z 346.084,A -85,B 0,C 180,E1 -4177.033,E2 -4177.033} C_VEL
LIN {X 0,Y 531.191,Z 336.468,A -85,B 0,C 180,E1 -4178.089,E2 -4178.089} C_VEL
LIN {X 0,Y 531.371,Z 326.504,A -85,B 0,C 180,E1 -4178.981,E2 -4178.981} C_VEL
LIN {X 0,Y 531.639,Z 315.028,A -85,B 0,C 180,E1 -4179.8,E2 -4179.8} C_VEL
LIN {X 0,Y 531.935,Z 302.92,A -85,B 0,C 180,E1 -4180.47,E2 -4180.47} C_VEL
LIN {X 0,Y 532.117,Z 291.449,A -85,B 0,C 180,E1 -4180.953,E2 -4180.953} C_VEL
LIN {X 0,Y 532.334,Z 278.354,A -85,B 0,C 180,E1 -4181.34,E2 -4181.34} C_VEL
LIN {X 0,Y 532.424,Z 262.041,A -85,B 0,C 180,E1 -4181.616,E2 -4181.616} C_VEL
LIN {X 0,Y 532.693,Z 175.167,A -85,B 0,C 180,E1 -4182.821,E2 -4182.821} C_VEL
LIN {X 0,Y 531.273,Z 166.781,A -85,B 0,C 180,E1 -4183.004,E2 -4183.004} C_VEL
LIN {X 0,Y 531.58,Z 148.938,A -85,B 0,C 180,E1 -4186.32,E2 -4186.32} C_VEL
LIN {X 0,Y 531.587,Z 141.277,A -85,B 0,C 180,E1 -4187.763,E2 -4187.763} C_VEL
LIN {X 0,Y 531.023,Z 137.343,A -85,B 0,C 180,E1 -4188.567,E2 -4188.567} C_VEL
LIN {X 0,Y 530.954,Z 137.343,A -85,B 0,C 180,E1 -4191.528,E2 -4191.528} C_VEL
LIN {X 0,Y 530.94,Z 137.351,A -85,B 0,C 180,E1 -4194.378,E2 -4194.378} C_VEL
LIN {X 0,Y 530.97,Z 137.341,A -85,B 0,C 180,E1 -4197.133,E2 -4197.133} C_VEL
LIN {X 0,Y 530.936,Z 137.345,A -85,B 0,C 180,E1 -4199.8,E2 -4199.8} C_VEL
LIN {X 0,Y 530.964,Z 137.348,A -85,B 0,C 180,E1 -4202.479,E2 -4202.479} C_VEL
LIN {X 0,Y 530.945,Z 137.344,A -85,B 0,C 180,E1 -4204.939,E2 -4204.939} C_VEL
LIN {X 0,Y 530.964,Z 137.344,A -85,B 0,C 180,E1 -4207.903,E2 -4207.903} C_VEL
LIN {X 0,Y 530.944,Z 137.346,A -85,B 0,C 180,E1 -4210.675,E2 -4210.675} C_VEL
LIN {X 0,Y 530.933,Z 137.344,A -85,B 0,C 180,E1 -4213.069,E2 -4213.069} C_VEL
LIN {X 0,Y 531.004,Z 137.337,A -85,B 0,C 180,E1 -4215.435,E2 -4215.435} C_VEL
LIN {X 0,Y 530.992,Z 137.339,A -85,B 0,C 180,E1 -4218.548,E2 -4218.548} C_VEL
LIN {X 0,Y 530.987,Z 137.342,A -85,B 0,C 180,E1 -4221.628,E2 -4221.628} C_VEL
LIN {X 0,Y 531.086,Z 137.326,A -85,B 0,C 180,E1 -4224.684,E2 -4224.684} C_VEL
LIN {X 0,Y 531.137,Z 137.326,A -85,B 0,C 180,E1 -4227.724,E2 -4227.724} C_VEL
LIN {X 0,Y 531.132,Z 137.326,A -85,B 0,C 180,E1 -4229.999,E2 -4229.999} C_VEL
LIN {X 0,Y 531.136,Z 137.321,A -85,B 0,C 180,E1 -4232.274,E2 -4232.274} C_VEL
LIN {X 0,Y 531.084,Z 137.329,A -85,B 0,C 180,E1 -4235.314,E2 -4235.314} C_VEL
LIN {X 0,Y 530.986,Z 137.338,A -85,B 0,C 180,E1 -4238.371,E2 -4238.371} C_VEL
LIN {X 0,Y 531.014,Z 137.342,A -85,B 0,C 180,E1 -4241.649,E2 -4241.649} C_VEL
LIN {X 0,Y 531.021,Z 137.335,A -85,B 0,C 180,E1 -4244.949,E2 -4244.949} C_VEL
LIN {X 0,Y 530.973,Z 137.344,A -85,B 0,C 180,E1 -4247.723,E2 -4247.723} C_VEL
LIN {X 0,Y 530.973,Z 137.34,A -85,B 0,C 180,E1 -4250.128,E2 -4250.128} C_VEL
LIN {X 0,Y 530.918,Z 137.347,A -85,B 0,C 180,E1 -4252.574,E2 -4252.574} C_VEL
LIN {X 0,Y 530.946,Z 137.349,A -85,B 0,C 180,E1 -4255.06,E2 -4255.06} C_VEL
LIN {X 0,Y 530.951,Z 137.346,A -85,B 0,C 180,E1 -4257.598,E2 -4257.598} C_VEL
LIN {X 0,Y 530.928,Z 137.345,A -85,B 0,C 180,E1 -4260.199,E2 -4260.199} C_VEL
LIN {X 0,Y 530.963,Z 137.346,A -85,B 0,C 180,E1 -4262.866,E2 -4262.866} C_VEL
LIN {X 0,Y 530.932,Z 137.346,A -85,B 0,C 180,E1 -4265.621,E2 -4265.621} C_VEL
LIN {X 0,Y 530.959,Z 137.345,A -85,B 0,C 180,E1 -4268.652,E2 -4268.652} C_VEL
LIN {X 0,Y 530.949,Z 137.345,A -85,B 0,C 180,E1 -4271.439,E2 -4271.439} C_VEL
LIN {X 0,Y 530.96,Z 137.345,A -85,B 0,C 180,E1 -4274.549,E2 -4274.549} C_VEL
LIN {X 0,Y 530.91,Z 137.348,A -85,B 0,C 180,E1 -4277.536,E2 -4277.536} C_VEL
LIN {X 0,Y 530.96,Z 137.347,A -85,B 0,C 180,E1 -4280.554,E2 -4280.554} C_VEL
LIN {X 0,Y 530.938,Z 137.344,A -85,B 0,C 180,E1 -4283.44,E2 -4283.44} C_VEL
LIN {X 0,Y 530.955,Z 137.349,A -85,B 0,C 180,E1 -4286.5,E2 -4286.5} C_VEL
LIN {X 0,Y 530.942,Z 137.344,A -85,B 0,C 180,E1 -4289.359,E2 -4289.359} C_VEL
LIN {X 0,Y 530.944,Z 137.351,A -85,B 0,C 180,E1 -4292.4,E2 -4292.4} C_VEL
LIN {X 0,Y 530.942,Z 137.346,A -85,B 0,C 180,E1 -4294.939,E2 -4294.939} C_VEL
LIN {X 0,Y 530.944,Z 137.35,A -85,B 0,C 180,E1 -4298.245,E2 -4298.245} C_VEL
LIN {X 0,Y 530.955,Z 137.346,A -85,B 0,C 180,E1 -4300.675,E2 -4300.675} C_VEL
LIN {X 0,Y 530.929,Z 137.345,A -85,B 0,C 180,E1 -4303.069,E2 -4303.069} C_VEL
LIN {X 0,Y 530.99,Z 137.338,A -85,B 0,C 180,E1 -4305.435,E2 -4305.435} C_VEL
LIN {X 0,Y 530.978,Z 137.343,A -85,B 0,C 180,E1 -4308.548,E2 -4308.548} C_VEL
LIN {X 0,Y 530.975,Z 137.342,A -85,B 0,C 180,E1 -4311.628,E2 -4311.628} C_VEL
LIN {X 0,Y 531.078,Z 137.328,A -85,B 0,C 180,E1 -4314.685,E2 -4314.685} C_VEL
LIN {X 0,Y 531.126,Z 137.326,A -85,B 0,C 180,E1 -4317.725,E2 -4317.725} C_VEL
LIN {X 0,Y 531.12,Z 137.33,A -85,B 0,C 180,E1 -4320,E2 -4320} C_VEL
LIN {X 0,Y 531.126,Z 137.324,A -85,B 0,C 180,E1 -4322.275,E2 -4322.275} C_VEL
LIN {X 0,Y 531.074,Z 137.329,A -85,B 0,C 180,E1 -4325.315,E2 -4325.315} C_VEL
LIN {X 0,Y 530.974,Z 137.341,A -85,B 0,C 180,E1 -4328.372,E2 -4328.372} C_VEL
LIN {X 0,Y 531.003,Z 137.344,A -85,B 0,C 180,E1 -4331.65,E2 -4331.65} C_VEL
LIN {X 0,Y 531.01,Z 137.336,A -85,B 0,C 180,E1 -4334.95,E2 -4334.95} C_VEL
LIN {X 0,Y 530.962,Z 137.348,A -85,B 0,C 180,E1 -4337.724,E2 -4337.724} C_VEL
LIN {X 0,Y 530.963,Z 137.342,A -85,B 0,C 180,E1 -4340.13,E2 -4340.13} C_VEL
LIN {X 0,Y 530.908,Z 137.348,A -85,B 0,C 180,E1 -4342.575,E2 -4342.575} C_VEL
LIN {X 0,Y 530.936,Z 137.348,A -85,B 0,C 180,E1 -4345.061,E2 -4345.061} C_VEL
LIN {X 0,Y 530.942,Z 137.349,A -85,B 0,C 180,E1 -4347.6,E2 -4347.6} C_VEL
LIN {X 0,Y 530.934,Z 137.345,A -85,B 0,C 180,E1 -4350.639,E2 -4350.639} C_VEL
LIN {X 0,Y 530.953,Z 137.347,A -85,B 0,C 180,E1 -4353.5,E2 -4353.5} C_VEL
LIN {X 0,Y 530.901,Z 137.348,A -85,B 0,C 180,E1 -4356.148,E2 -4356.148} C_VEL
LIN {X 0,Y 530.948,Z 137.345,A -85,B 0,C 180,E1 -4358.652,E2 -4358.652} C_VEL
LIN {X 0,Y 530.944,Z 137.347,A -85,B 0,C 180,E1 -4361.44,E2 -4361.44} C_VEL
LIN {X 0,Y 530.957,Z 137.344,A -85,B 0,C 180,E1 -4364.55,E2 -4364.55} C_VEL
LIN {X 0,Y 530.906,Z 137.349,A -85,B 0,C 180,E1 -4367.537,E2 -4367.537} C_VEL
LIN {X 0,Y 530.948,Z 137.347,A -85,B 0,C 180,E1 -4370.554,E2 -4370.554} C_VEL
LIN {X 0,Y 530.902,Z 137.35,A -85,B 0,C 180,E1 -4373.438,E2 -4373.438} C_VEL
LIN {X 0,Y 530.945,Z 137.345,A -85,B 0,C 180,E1 -4376.225,E2 -4376.225} C_VEL
LIN {X 0,Y 530.931,Z 137.351,A -85,B 0,C 180,E1 -4378.92,E2 -4378.92} C_VEL
LIN {X 0,Y 530.926,Z 137.346,A -85,B 0,C 180,E1 -4381.541,E2 -4381.541} C_VEL
LIN {X 0,Y 530.957,Z 137.347,A -85,B 0,C 180,E1 -4384.169,E2 -4384.169} C_VEL
LIN {X 0,Y 530.953,Z 137.374,A -85,B 0,C 180,E1 -4386.016,E2 -4386.016} C_VEL
LIN {X 0,Y 532.219,Z 144.796,A -85,B 0,C 180,E1 -4387.28,E2 -4387.28} C_VEL
LIN {X 0,Y 531.954,Z 161.269,A -85,B 0,C 180,E1 -4389.91,E2 -4389.91} C_VEL
LIN {X 0,Y 531.534,Z 180.293,A -85,B 0,C 180,E1 -4392.892,E2 -4392.892} C_VEL
LIN {X 0,Y 531.278,Z 194.304,A -85,B 0,C 180,E1 -4395.058,E2 -4395.058} C_VEL
LIN {X 0,Y 532.724,Z 205.026,A -85,B 0,C 180,E1 -4395.252,E2 -4395.252} C_VEL
LIN {X 0,Y 532.367,Z 301.805,A -85,B 0,C 180,E1 -4396.595,E2 -4396.595} C_VEL
LIN {X 0,Y 532.155,Z 315.225,A -85,B 0,C 180,E1 -4396.929,E2 -4396.929} C_VEL
LIN {X 0,Y 531.931,Z 328.031,A -85,B 0,C 180,E1 -4397.409,E2 -4397.409} C_VEL
LIN {X 0,Y 531.662,Z 339.934,A -85,B 0,C 180,E1 -4398.015,E2 -4398.015} C_VEL
LIN {X 0,Y 531.476,Z 351.145,A -85,B 0,C 180,E1 -4398.753,E2 -4398.753} C_VEL
LIN {X 0,Y 531.208,Z 361.683,A -85,B 0,C 180,E1 -4399.616,E2 -4399.616} C_VEL
LIN {X 0,Y 530.986,Z 370.294,A -85,B 0,C 180,E1 -4400.478,E2 -4400.478} C_VEL
LIN {X 0,Y 530.847,Z 378.236,A -85,B 0,C 180,E1 -4401.435,E2 -4401.435} C_VEL
LIN {X 0,Y 530.666,Z 385.988,A -85,B 0,C 180,E1 -4402.582,E2 -4402.582} C_VEL
LIN {X 0,Y 530.574,Z 393.117,A -85,B 0,C 180,E1 -4403.918,E2 -4403.918} C_VEL
LIN {X 0,Y 530.459,Z 397.86,A -85,B 0,C 180,E1 -4405.06,E2 -4405.06} C_VEL
LIN {X 0,Y 530.516,Z 401.485,A -85,B 0,C 180,E1 -4406.203,E2 -4406.203} C_VEL
LIN {X 0,Y 530.457,Z 403.353,A -85,B 0,C 180,E1 -4406.963,E2 -4406.963} C_VEL
LIN {X 0,Y 530.411,Z 404.752,A -85,B 0,C 180,E1 -4407.723,E2 -4407.723} C_VEL
LIN {X 0,Y 530.347,Z 406.357,A -85,B 0,C 180,E1 -4409.241,E2 -4409.241} C_VEL
LIN {X 0,Y 530.348,Z 406.572,A -85,B 0,C 180,E1 -4410.001,E2 -4410.001} C_VEL
LIN {X 0,Y 530.361,Z 405.742,A -85,B 0,C 180,E1 -4411.519,E2 -4411.519} C_VEL
LIN {X 0,Y 530.411,Z 404.742,A -85,B 0,C 180,E1 -4412.279,E2 -4412.279} C_VEL
LIN {X 0,Y 530.457,Z 403.337,A -85,B 0,C 180,E1 -4413.038,E2 -4413.038} C_VEL
LIN {X 0,Y 530.521,Z 400.386,A -85,B 0,C 180,E1 -4414.179,E2 -4414.179} C_VEL
LIN {X 0,Y 530.522,Z 396.386,A -85,B 0,C 180,E1 -4415.321,E2 -4415.321} C_VEL
LIN {X 0,Y 530.583,Z 390.705,A -85,B 0,C 180,E1 -4416.567,E2 -4416.567} C_VEL
LIN {X 0,Y 530.705,Z 383.506,A -85,B 0,C 180,E1 -4417.802,E2 -4417.802} C_VEL
LIN {X 0,Y 530.881,Z 375.15,A -85,B 0,C 180,E1 -4418.949,E2 -4418.949} C_VEL
LIN {X 0,Y 531.058,Z 366.562,A -85,B 0,C 180,E1 -4419.907,E2 -4419.907} C_VEL
LIN {X 0,Y 531.312,Z 355.957,A -85,B 0,C 180,E1 -4420.866,E2 -4420.866} C_VEL
LIN {X 0,Y 531.583,Z 344.208,A -85,B 0,C 180,E1 -4421.715,E2 -4421.715} C_VEL
LIN {X 0,Y 531.846,Z 331.873,A -85,B 0,C 180,E1 -4422.4,E2 -4422.4} C_VEL
LIN {X 0,Y 532.072,Z 319.242,A -85,B 0,C 180,E1 -4422.928,E2 -4422.928} C_VEL
LIN {X 0,Y 532.244,Z 306.992,A -85,B 0,C 180,E1 -4423.288,E2 -4423.288} C_VEL
LIN {X 0,Y 532.416,Z 291.611,A -85,B 0,C 180,E1 -4423.551,E2 -4423.551} C_VEL
LIN {X 0,Y 532.711,Z 203.807,A -85,B 0,C 180,E1 -4424.762,E2 -4424.762} C_VEL
LIN {X 0,Y 531.254,Z 193.793,A -85,B 0,C 180,E1 -4424.962,E2 -4424.962} C_VEL
LIN {X 0,Y 531.524,Z 175.135,A -85,B 0,C 180,E1 -4427.822,E2 -4427.822} C_VEL
LIN {X 0,Y 531.9,Z 157.739,A -85,B 0,C 180,E1 -4430.513,E2 -4430.513} C_VEL
LIN {X 0,Y 532.026,Z 143.572,A -85,B 0,C 180,E1 -4432.731,E2 -4432.731} C_VEL
LIN {X 0,Y 530.962,Z 137.349,A -85,B 0,C 180,E1 -4433.759,E2 -4433.759} C_VEL
LIN {X 0,Y 530.944,Z 137.349,A -85,B 0,C 180,E1 -4436.748,E2 -4436.748} C_VEL
LIN {X 0,Y 530.918,Z 137.356,A -85,B 0,C 180,E1 -4439.327,E2 -4439.327} C_VEL
LIN {X 0,Y 530.955,Z 137.344,A -85,B 0,C 180,E1 -4442.098,E2 -4442.098} C_VEL
LIN {X 0,Y 530.957,Z 137.348,A -85,B 0,C 180,E1 -4444.849,E2 -4444.849} C_VEL
LIN {X 0,Y 530.935,Z 137.348,A -85,B 0,C 180,E1 -4447.511,E2 -4447.511} C_VEL
LIN {X 0,Y 530.948,Z 137.346,A -85,B 0,C 180,E1 -4450.437,E2 -4450.437} C_VEL
LIN {X 0,Y 530.929,Z 137.346,A -85,B 0,C 180,E1 -4453.499,E2 -4453.499} C_VEL
LIN {X 0,Y 530.968,Z 137.34,A -85,B 0,C 180,E1 -4455.624,E2 -4455.624} C_VEL
LIN {X 0,Y 530.933,Z 137.349,A -85,B 0,C 180,E1 -4458.984,E2 -4458.984} C_VEL
LIN {X 0,Y 530.951,Z 137.342,A -85,B 0,C 180,E1 -4461.529,E2 -4461.529} C_VEL
LIN {X 0,Y 530.937,Z 137.349,A -85,B 0,C 180,E1 -4464.379,E2 -4464.379} C_VEL
LIN {X 0,Y 530.968,Z 137.342,A -85,B 0,C 180,E1 -4467.133,E2 -4467.133} C_VEL
LIN {X 0,Y 530.936,Z 137.345,A -85,B 0,C 180,E1 -4469.801,E2 -4469.801} C_VEL
LIN {X 0,Y 530.957,Z 137.349,A -85,B 0,C 180,E1 -4472.48,E2 -4472.48} C_VEL
LIN {X 0,Y 530.952,Z 137.344,A -85,B 0,C 180,E1 -4474.94,E2 -4474.94} C_VEL
LIN {X 0,Y 530.979,Z 137.343,A -85,B 0,C 180,E1 -4477.899,E2 -4477.899} C_VEL
LIN {X 0,Y 530.972,Z 137.342,A -85,B 0,C 180,E1 -4480.676,E2 -4480.676} C_VEL
LIN {X 0,Y 530.932,Z 137.346,A -85,B 0,C 180,E1 -4483.069,E2 -4483.069} C_VEL
LIN {X 0,Y 531.016,Z 137.337,A -85,B 0,C 180,E1 -4485.436,E2 -4485.436} C_VEL
LIN {X 0,Y 531.038,Z 137.335,A -85,B 0,C 180,E1 -4488.55,E2 -4488.55} C_VEL
LIN {X 0,Y 530.994,Z 137.345,A -85,B 0,C 180,E1 -4491.629,E2 -4491.629} C_VEL
LIN {X 0,Y 531.093,Z 137.326,A -85,B 0,C 180,E1 -4494.685,E2 -4494.685} C_VEL
LIN {X 0,Y 531.138,Z 137.328,A -85,B 0,C 180,E1 -4497.725,E2 -4497.725} C_VEL
LIN {X 0,Y 531.135,Z 137.326,A -85,B 0,C 180,E1 -4500,E2 -4500} C_VEL
LIN {X 0,Y 531.096,Z 137.33,A -85,B 0,C 180,E1 -4503.034,E2 -4503.034} C_VEL
LIN {X 0,Y 531.054,Z 137.336,A -85,B 0,C 180,E1 -4506.078,E2 -4506.078} C_VEL
LIN {X 0,Y 531.07,Z 137.381,A -85,B 0,C 180,E1 -4507.94,E2 -4507.94} C_VEL
LIN {X 0,Y 531.431,Z 141.93,A -85,B 0,C 180,E1 -4508.748,E2 -4508.748} C_VEL
LIN {X 0,Y 531.361,Z 156.36,A -85,B 0,C 180,E1 -4511.25,E2 -4511.25} C_VEL
LIN {X 0,Y 531.23,Z 166.835,A -85,B 0,C 180,E1 -4513.095,E2 -4513.095} C_VEL
LIN {X 0,Y 532.824,Z 176.827,A -85,B 0,C 180,E1 -4513.297,E2 -4513.297} C_VEL
LIN {X 0,Y 532.373,Z 274.551,A -85,B 0,C 180,E1 -4514.673,E2 -4514.673} C_VEL
LIN {X 0,Y 532.19,Z 287.158,A -85,B 0,C 180,E1 -4514.996,E2 -4514.996} C_VEL
LIN {X 0,Y 532.008,Z 299.507,A -85,B 0,C 180,E1 -4515.462,E2 -4515.462} C_VEL
LIN {X 0,Y 531.749,Z 312.154,A -85,B 0,C 180,E1 -4516.114,E2 -4516.114} C_VEL
LIN {X 0,Y 531.455,Z 324.024,A -85,B 0,C 180,E1 -4516.914,E2 -4516.914} C_VEL
LIN {X 0,Y 531.26,Z 333.756,A -85,B 0,C 180,E1 -4517.732,E2 -4517.732} C_VEL
LIN {X 0,Y 531.035,Z 343.268,A -85,B 0,C 180,E1 -4518.72,E2 -4518.72} C_VEL
LIN {X 0,Y 530.846,Z 350.789,A -85,B 0,C 180,E1 -4519.667,E2 -4519.667} C_VEL
LIN {X 0,Y 530.707,Z 359.003,A -85,B 0,C 180,E1 -4520.95,E2 -4520.95} C_VEL
LIN {X 0,Y 530.567,Z 365.507,A -85,B 0,C 180,E1 -4522.254,E2 -4522.254} C_VEL
LIN {X 0,Y 530.508,Z 369.969,A -85,B 0,C 180,E1 -4523.418,E2 -4523.418} C_VEL
LIN {X 0,Y 530.477,Z 372.163,A -85,B 0,C 180,E1 -4524.134,E2 -4524.134} C_VEL
LIN {X 0,Y 529.821,Z 373.763,A -85,B 0,C 180,E1 -4524.744,E2 -4524.744} C_VEL
LIN {X 0,Y 526.908,Z 375.809,A -85,B 0,C 180,E1 -4525.748,E2 -4525.748} C_VEL
LIN {X 0,Y 524.43,Z 376.909,A -85,B 0,C 180,E1 -4526.566,E2 -4526.566} C_VEL
LIN {X 0,Y 523.363,Z 377.446,A -85,B 0,C 180,E1 -4527.204,E2 -4527.204} C_VEL
LIN {X 0,Y 523.276,Z 377.541,A -85,B 0,C 180,E1 -4527.42,E2 -4527.42} C_VEL
LIN {X 0,Y 523.288,Z 377.7,A -85,B 0,C 180,E1 -4528.039,E2 -4528.039} C_VEL
LIN {X 0,Y 523.325,Z 377.242,A -85,B 0,C 180,E1 -4529.2,E2 -4529.2} C_VEL
LIN {X 0,Y 523.361,Z 375.207,A -85,B 0,C 180,E1 -4530.747,E2 -4530.747} C_VEL
LIN {X 0,Y 523.404,Z 371.708,A -85,B 0,C 180,E1 -4532.227,E2 -4532.227} C_VEL
LIN {X 0,Y 523.439,Z 367.727,A -85,B 0,C 180,E1 -4533.401,E2 -4533.401} C_VEL
LIN {X 0,Y 523.535,Z 362.073,A -85,B 0,C 180,E1 -4534.68,E2 -4534.68} C_VEL
LIN {X 0,Y 523.709,Z 354.802,A -85,B 0,C 180,E1 -4535.953,E2 -4535.953} C_VEL
LIN {X 0,Y 523.922,Z 346.388,A -85,B 0,C 180,E1 -4537.132,E2 -4537.132} C_VEL
LIN {X 0,Y 524.179,Z 336.801,A -85,B 0,C 180,E1 -4538.202,E2 -4538.202} C_VEL
LIN {X 0,Y 524.428,Z 326.131,A -85,B 0,C 180,E1 -4539.164,E2 -4539.164} C_VEL
LIN {X 0,Y 524.654,Z 316.146,A -85,B 0,C 180,E1 -4539.89,E2 -4539.89} C_VEL
LIN {X 0,Y 524.971,Z 304.278,A -85,B 0,C 180,E1 -4540.57,E2 -4540.57} C_VEL
LIN {X 0,Y 525.191,Z 291.495,A -85,B 0,C 180,E1 -4541.122,E2 -4541.122} C_VEL
LIN {X 0,Y 525.406,Z 278.964,A -85,B 0,C 180,E1 -4541.5,E2 -4541.5} C_VEL
LIN {X 0,Y 525.519,Z 263.83,A -85,B 0,C 180,E1 -4541.767,E2 -4541.767} C_VEL
LIN {X 0,Y 525.817,Z 175.825,A -85,B 0,C 180,E1 -4543.01,E2 -4543.01} C_VEL
LIN {X 0,Y 524.268,Z 166.976,A -85,B 0,C 180,E1 -4543.204,E2 -4543.204} C_VEL
LIN {X 0,Y 524.584,Z 150.236,A -85,B 0,C 180,E1 -4546.341,E2 -4546.341} C_VEL
LIN {X 0,Y 524.671,Z 143.128,A -85,B 0,C 180,E1 -4547.696,E2 -4547.696} C_VEL
LIN {X 0,Y 523.968,Z 138.222,A -85,B 0,C 180,E1 -4548.689,E2 -4548.689} C_VEL
LIN {X 0,Y 523.915,Z 138.221,A -85,B 0,C 180,E1 -4551.898,E2 -4551.898} C_VEL
LIN {X 0,Y 523.92,Z 138.222,A -85,B 0,C 180,E1 -4554.913,E2 -4554.913} C_VEL
LIN {X 0,Y 523.936,Z 138.216,A -85,B 0,C 180,E1 -4557.681,E2 -4557.681} C_VEL
LIN {X 0,Y 523.885,Z 138.227,A -85,B 0,C 180,E1 -4560.691,E2 -4560.691} C_VEL
LIN {X 0,Y 523.901,Z 138.223,A -85,B 0,C 180,E1 -4562.864,E2 -4562.864} C_VEL
LIN {X 0,Y 523.916,Z 138.221,A -85,B 0,C 180,E1 -4565.809,E2 -4565.809} C_VEL
LIN {X 0,Y 523.909,Z 138.222,A -85,B 0,C 180,E1 -4568.764,E2 -4568.764} C_VEL
LIN {X 0,Y 523.917,Z 138.218,A -85,B 0,C 180,E1 -4571.219,E2 -4571.219} C_VEL
LIN {X 0,Y 523.905,Z 138.225,A -85,B 0,C 180,E1 -4574.437,E2 -4574.437} C_VEL
LIN {X 0,Y 523.935,Z 138.217,A -85,B 0,C 180,E1 -4576.818,E2 -4576.818} C_VEL
LIN {X 0,Y 523.938,Z 138.216,A -85,B 0,C 180,E1 -4579.175,E2 -4579.175} C_VEL
LIN {X 0,Y 523.955,Z 138.218,A -85,B 0,C 180,E1 -4582.291,E2 -4582.291} C_VEL
LIN {X 0,Y 524.033,Z 138.205,A -85,B 0,C 180,E1 -4584.613,E2 -4584.613} C_VEL
LIN {X 0,Y 524.108,Z 138.201,A -85,B 0,C 180,E1 -4587.694,E2 -4587.694} C_VEL
LIN {X 0,Y 524.1,Z 138.202,A -85,B 0,C 180,E1 -4589.999,E2 -4589.999} C_VEL
LIN {X 0,Y 524.106,Z 138.197,A -85,B 0,C 180,E1 -4592.305,E2 -4592.305} C_VEL
LIN {X 0,Y 524.001,Z 138.211,A -85,B 0,C 180,E1 -4596.159,E2 -4596.159} C_VEL
LIN {X 0,Y 523.947,Z 138.219,A -85,B 0,C 180,E1 -4599.262,E2 -4599.262} C_VEL
LIN {X 0,Y 523.93,Z 138.217,A -85,B 0,C 180,E1 -4602.393,E2 -4602.393} C_VEL
LIN {X 0,Y 523.914,Z 138.227,A -85,B 0,C 180,E1 -4605.562,E2 -4605.562} C_VEL
LIN {X 0,Y 523.912,Z 138.221,A -85,B 0,C 180,E1 -4607.97,E2 -4607.97} C_VEL
LIN {X 0,Y 523.917,Z 138.218,A -85,B 0,C 180,E1 -4610.411,E2 -4610.411} C_VEL
LIN {X 0,Y 523.886,Z 138.225,A -85,B 0,C 180,E1 -4612.894,E2 -4612.894} C_VEL
LIN {X 0,Y 523.897,Z 138.228,A -85,B 0,C 180,E1 -4615.421,E2 -4615.421} C_VEL
LIN {X 0,Y 523.896,Z 138.222,A -85,B 0,C 180,E1 -4618.002,E2 -4618.002} C_VEL
LIN {X 0,Y 523.897,Z 138.225,A -85,B 0,C 180,E1 -4620.845,E2 -4620.845} C_VEL
LIN {X 0,Y 523.925,Z 138.219,A -85,B 0,C 180,E1 -4623.728,E2 -4623.728} C_VEL
LIN {X 0,Y 523.885,Z 138.224,A -85,B 0,C 180,E1 -4626.398,E2 -4626.398} C_VEL
LIN {X 0,Y 523.908,Z 138.227,A -85,B 0,C 180,E1 -4629.085,E2 -4629.085} C_VEL
LIN {X 0,Y 523.89,Z 138.222,A -85,B 0,C 180,E1 -4632.124,E2 -4632.124} C_VEL
LIN {X 0,Y 523.93,Z 138.22,A -85,B 0,C 180,E1 -4635.31,E2 -4635.31} C_VEL
LIN {X 0,Y 523.907,Z 138.227,A -85,B 0,C 180,E1 -4638.695,E2 -4638.695} C_VEL
LIN {X 0,Y 523.905,Z 138.22,A -85,B 0,C 180,E1 -4641.897,E2 -4641.897} C_VEL
LIN {X 0,Y 523.909,Z 138.225,A -85,B 0,C 180,E1 -4644.912,E2 -4644.912} C_VEL
LIN {X 0,Y 523.925,Z 138.217,A -85,B 0,C 180,E1 -4647.68,E2 -4647.68} C_VEL
LIN {X 0,Y 523.924,Z 138.225,A -85,B 0,C 180,E1 -4650.681,E2 -4650.681} C_VEL
LIN {X 0,Y 523.892,Z 138.222,A -85,B 0,C 180,E1 -4653.724,E2 -4653.724} C_VEL
LIN {X 0,Y 523.89,Z 138.228,A -85,B 0,C 180,E1 -4656.268,E2 -4656.268} C_VEL
LIN {X 0,Y 523.916,Z 138.222,A -85,B 0,C 180,E1 -4658.765,E2 -4658.765} C_VEL
LIN {X 0,Y 523.918,Z 138.218,A -85,B 0,C 180,E1 -4661.219,E2 -4661.219} C_VEL
LIN {X 0,Y 523.904,Z 138.226,A -85,B 0,C 180,E1 -4664.437,E2 -4664.437} C_VEL
LIN {X 0,Y 523.938,Z 138.217,A -85,B 0,C 180,E1 -4667.606,E2 -4667.606} C_VEL
LIN {X 0,Y 523.937,Z 138.217,A -85,B 0,C 180,E1 -4670.737,E2 -4670.737} C_VEL
LIN {X 0,Y 524.001,Z 138.214,A -85,B 0,C 180,E1 -4673.84,E2 -4673.84} C_VEL
LIN {X 0,Y 524.096,Z 138.201,A -85,B 0,C 180,E1 -4677.694,E2 -4677.694} C_VEL
LIN {X 0,Y 524.089,Z 138.205,A -85,B 0,C 180,E1 -4680,E2 -4680} C_VEL
LIN {X 0,Y 524.096,Z 138.199,A -85,B 0,C 180,E1 -4682.305,E2 -4682.305} C_VEL
LIN {X 0,Y 523.993,Z 138.213,A -85,B 0,C 180,E1 -4686.16,E2 -4686.16} C_VEL
LIN {X 0,Y 523.936,Z 138.219,A -85,B 0,C 180,E1 -4689.263,E2 -4689.263} C_VEL
LIN {X 0,Y 523.935,Z 138.217,A -85,B 0,C 180,E1 -4692.393,E2 -4692.393} C_VEL
LIN {X 0,Y 523.903,Z 138.229,A -85,B 0,C 180,E1 -4695.563,E2 -4695.563} C_VEL
LIN {X 0,Y 523.901,Z 138.224,A -85,B 0,C 180,E1 -4697.971,E2 -4697.971} C_VEL
LIN {X 0,Y 523.907,Z 138.22,A -85,B 0,C 180,E1 -4700.413,E2 -4700.413} C_VEL
LIN {X 0,Y 523.876,Z 138.225,A -85,B 0,C 180,E1 -4702.895,E2 -4702.895} C_VEL
LIN {X 0,Y 523.888,Z 138.231,A -85,B 0,C 180,E1 -4705.422,E2 -4705.422} C_VEL
LIN {X 0,Y 523.888,Z 138.223,A -85,B 0,C 180,E1 -4708.004,E2 -4708.004} C_VEL
LIN {X 0,Y 523.89,Z 138.225,A -85,B 0,C 180,E1 -4710.846,E2 -4710.846} C_VEL
LIN {X 0,Y 523.918,Z 138.221,A -85,B 0,C 180,E1 -4713.729,E2 -4713.729} C_VEL
LIN {X 0,Y 523.86,Z 138.226,A -85,B 0,C 180,E1 -4716.396,E2 -4716.396} C_VEL
LIN {X 0,Y 523.896,Z 138.23,A -85,B 0,C 180,E1 -4719.087,E2 -4719.087} C_VEL
LIN {X 0,Y 523.886,Z 138.222,A -85,B 0,C 180,E1 -4722.126,E2 -4722.126} C_VEL
LIN {X 0,Y 523.928,Z 138.222,A -85,B 0,C 180,E1 -4725.312,E2 -4725.312} C_VEL
LIN {X 0,Y 523.903,Z 138.226,A -85,B 0,C 180,E1 -4728.697,E2 -4728.697} C_VEL
LIN {X 0,Y 523.9,Z 138.227,A -85,B 0,C 180,E1 -4731.083,E2 -4731.083} C_VEL
LIN {X 0,Y 523.851,Z 138.227,A -85,B 0,C 180,E1 -4733.822,E2 -4733.822} C_VEL
LIN {X 0,Y 523.906,Z 138.227,A -85,B 0,C 180,E1 -4736.634,E2 -4736.634} C_VEL
LIN {X 0,Y 523.903,Z 138.222,A -85,B 0,C 180,E1 -4739.353,E2 -4739.353} C_VEL
LIN {X 0,Y 523.908,Z 138.224,A -85,B 0,C 180,E1 -4742.296,E2 -4742.296} C_VEL
LIN {X 0,Y 523.896,Z 138.227,A -85,B 0,C 180,E1 -4745.427,E2 -4745.427} C_VEL
LIN {X 0,Y 523.915,Z 138.268,A -85,B 0,C 180,E1 -4745.847,E2 -4745.847} C_VEL
LIN {X 0,Y 525.265,Z 145.919,A -85,B 0,C 180,E1 -4747.17,E2 -4747.17} C_VEL
LIN {X 0,Y 524.979,Z 162.378,A -85,B 0,C 180,E1 -4749.836,E2 -4749.836} C_VEL
LIN {X 0,Y 524.549,Z 178.85,A -85,B 0,C 180,E1 -4752.456,E2 -4752.456} C_VEL
LIN {X 0,Y 524.278,Z 194.137,A -85,B 0,C 180,E1 -4754.854,E2 -4754.854} C_VEL
LIN {X 0,Y 525.857,Z 204.874,A -85,B 0,C 180,E1 -4755.056,E2 -4755.056} C_VEL
LIN {X 0,Y 525.433,Z 302.395,A -85,B 0,C 180,E1 -4756.439,E2 -4756.439} C_VEL
LIN {X 0,Y 525.201,Z 315.528,A -85,B 0,C 180,E1 -4756.778,E2 -4756.778} C_VEL
LIN {X 0,Y 524.97,Z 328.756,A -85,B 0,C 180,E1 -4757.288,E2 -4757.288} C_VEL
LIN {X 0,Y 524.668,Z 340.651,A -85,B 0,C 180,E1 -4757.918,E2 -4757.918} C_VEL
LIN {X 0,Y 524.451,Z 352.139,A -85,B 0,C 180,E1 -4758.698,E2 -4758.698} C_VEL
LIN {X 0,Y 524.156,Z 362.47,A -85,B 0,C 180,E1 -4759.572,E2 -4759.572} C_VEL
LIN {X 0,Y 523.919,Z 371.741,A -85,B 0,C 180,E1 -4760.543,E2 -4760.543} C_VEL
LIN {X 0,Y 523.72,Z 380.752,A -85,B 0,C 180,E1 -4761.706,E2 -4761.706} C_VEL
LIN {X 0,Y 523.567,Z 388.008,A -85,B 0,C 180,E1 -4762.868,E2 -4762.868} C_VEL
LIN {X 0,Y 523.469,Z 392.899,A -85,B 0,C 180,E1 -4763.835,E2 -4763.835} C_VEL
LIN {X 0,Y 523.383,Z 397.651,A -85,B 0,C 180,E1 -4764.993,E2 -4764.993} C_VEL
LIN {X 0,Y 523.443,Z 401.283,A -85,B 0,C 180,E1 -4766.151,E2 -4766.151} C_VEL
LIN {X 0,Y 523.367,Z 403.154,A -85,B 0,C 180,E1 -4766.922,E2 -4766.922} C_VEL
LIN {X 0,Y 523.335,Z 404.556,A -85,B 0,C 180,E1 -4767.692,E2 -4767.692} C_VEL
LIN {X 0,Y 523.253,Z 406.163,A -85,B 0,C 180,E1 -4769.231,E2 -4769.231} C_VEL
LIN {X 0,Y 523.251,Z 406.377,A -85,B 0,C 180,E1 -4770.001,E2 -4770.001} C_VEL
LIN {X 0,Y 523.275,Z 405.545,A -85,B 0,C 180,E1 -4771.54,E2 -4771.54} C_VEL
LIN {X 0,Y 523.335,Z 404.541,A -85,B 0,C 180,E1 -4772.31,E2 -4772.31} C_VEL
LIN {X 0,Y 523.367,Z 403.131,A -85,B 0,C 180,E1 -4773.08,E2 -4773.08} C_VEL
LIN {X 0,Y 523.422,Z 400.171,A -85,B 0,C 180,E1 -4774.236,E2 -4774.236} C_VEL
LIN {X 0,Y 523.456,Z 396.162,A -85,B 0,C 180,E1 -4775.393,E2 -4775.393} C_VEL
LIN {X 0,Y 523.501,Z 390.962,A -85,B 0,C 180,E1 -4776.56,E2 -4776.56} C_VEL
LIN {X 0,Y 523.628,Z 384.489,A -85,B 0,C 180,E1 -4777.714,E2 -4777.714} C_VEL
LIN {X 0,Y 523.789,Z 376.377,A -85,B 0,C 180,E1 -4778.877,E2 -4778.877} C_VEL
LIN {X 0,Y 523.974,Z 368.094,A -85,B 0,C 180,E1 -4779.847,E2 -4779.847} C_VEL
LIN {X 0,Y 524.285,Z 357.979,A -85,B 0,C 180,E1 -4780.817,E2 -4780.817} C_VEL
LIN {X 0,Y 524.521,Z 346.908,A -85,B 0,C 180,E1 -4781.666,E2 -4781.666} C_VEL
LIN {X 0,Y 524.818,Z 335.265,A -85,B 0,C 180,E1 -4782.373,E2 -4782.373} C_VEL
LIN {X 0,Y 525.056,Z 322.658,A -85,B 0,C 180,E1 -4782.957,E2 -4782.957} C_VEL
LIN {X 0,Y 525.298,Z 309.184,A -85,B 0,C 180,E1 -4783.393,E2 -4783.393} C_VEL
LIN {X 0,Y 525.497,Z 295.922,A -85,B 0,C 180,E1 -4783.659,E2 -4783.659} C_VEL
LIN {X 0,Y 525.759,Z 203.78,A -85,B 0,C 180,E1 -4784.959,E2 -4784.959} C_VEL
LIN {X 0,Y 524.227,Z 193.592,A -85,B 0,C 180,E1 -4785.164,E2 -4785.164} C_VEL
LIN {X 0,Y 524.57,Z 174.501,A -85,B 0,C 180,E1 -4788.13,E2 -4788.13} C_VEL
LIN {X 0,Y 524.958,Z 156.281,A -85,B 0,C 180,E1 -4790.985,E2 -4790.985} C_VEL
LIN {X 0,Y 525.031,Z 144.577,A -85,B 0,C 180,E1 -4792.843,E2 -4792.843} C_VEL
LIN {X 0,Y 523.903,Z 138.227,A -85,B 0,C 180,E1 -4793.939,E2 -4793.939} C_VEL
LIN {X 0,Y 523.894,Z 138.231,A -85,B 0,C 180,E1 -4797.137,E2 -4797.137} C_VEL
LIN {X 0,Y 523.868,Z 138.229,A -85,B 0,C 180,E1 -4799.761,E2 -4799.761} C_VEL
LIN {X 0,Y 523.902,Z 138.223,A -85,B 0,C 180,E1 -4802.452,E2 -4802.452} C_VEL
LIN {X 0,Y 523.909,Z 138.227,A -85,B 0,C 180,E1 -4805.228,E2 -4805.228} C_VEL
LIN {X 0,Y 523.903,Z 138.221,A -85,B 0,C 180,E1 -4808.104,E2 -4808.104} C_VEL
LIN {X 0,Y 523.917,Z 138.223,A -85,B 0,C 180,E1 -4811.305,E2 -4811.305} C_VEL
LIN {X 0,Y 523.936,Z 138.222,A -85,B 0,C 180,E1 -4814.689,E2 -4814.689} C_VEL
LIN {X 0,Y 523.894,Z 138.221,A -85,B 0,C 180,E1 -4817.875,E2 -4817.875} C_VEL
LIN {X 0,Y 523.912,Z 138.224,A -85,B 0,C 180,E1 -4820.914,E2 -4820.914} C_VEL
LIN {X 0,Y 523.881,Z 138.223,A -85,B 0,C 180,E1 -4823.824,E2 -4823.824} C_VEL
LIN {X 0,Y 523.915,Z 138.226,A -85,B 0,C 180,E1 -4826.634,E2 -4826.634} C_VEL
LIN {X 0,Y 523.915,Z 138.218,A -85,B 0,C 180,E1 -4829.353,E2 -4829.353} C_VEL
LIN {X 0,Y 523.914,Z 138.225,A -85,B 0,C 180,E1 -4832.296,E2 -4832.296} C_VEL
LIN {X 0,Y 523.905,Z 138.22,A -85,B 0,C 180,E1 -4835.427,E2 -4835.427} C_VEL
LIN {X 0,Y 523.94,Z 138.22,A -85,B 0,C 180,E1 -4837.94,E2 -4837.94} C_VEL
LIN {X 0,Y 523.959,Z 138.219,A -85,B 0,C 180,E1 -4840.407,E2 -4840.407} C_VEL
LIN {X 0,Y 523.899,Z 138.223,A -85,B 0,C 180,E1 -4842.835,E2 -4842.835} C_VEL
LIN {X 0,Y 523.977,Z 138.213,A -85,B 0,C 180,E1 -4845.236,E2 -4845.236} C_VEL
